LIN {X 0,Y 317.742,Z 934.096,A -85,B 0,C 180,E1 -15208.733,E2 -15208.733} C_VEL
LIN {X 0,Y 317.78,Z 934.392,A -85,B 0,C 180,E1 -15210,E2 -15210} C_VEL
LIN {X 0,Y 317.742,Z 934.092,A -85,B 0,C 180,E1 -15211.267,E2 -15211.267} C_VEL
LIN {X 0,Y 317.766,Z 933.304,A -85,B 0,C 180,E1 -15212.535,E2 -15212.535} C_VEL
LIN {X 0,Y 317.849,Z 932.043,A -85,B 0,C 180,E1 -15213.803,E2 -15213.803} C_VEL
LIN {X 0,Y 317.9,Z 930.281,A -85,B 0,C 180,E1 -15215.073,E2 -15215.073} C_VEL
LIN {X 0,Y 318.202,Z 926.465,A -85,B 0,C 180,E1 -15216.977,E2 -15216.977} C_VEL
LIN {X 0,Y 318.673,Z 921.267,A -85,B 0,C 180,E1 -15218.881,E2 -15218.881} C_VEL
LIN {X 0,Y 319.407,Z 914.42,A -85,B 0,C 180,E1 -15220.779,E2 -15220.779} C_VEL
LIN {X 0,Y 320.293,Z 906.941,A -85,B 0,C 180,E1 -15222.353,E2 -15222.353} C_VEL
LIN {X 0,Y 321.122,Z 899.567,A -85,B 0,C 180,E1 -15223.608,E2 -15223.608} C_VEL
LIN {X 0,Y 322.069,Z 891.674,A -85,B 0,C 180,E1 -15224.695,E2 -15224.695} C_VEL
LIN {X 0,Y 322.96,Z 883.333,A -85,B 0,C 180,E1 -15225.622,E2 -15225.622} C_VEL
LIN {X 0,Y 323.821,Z 872.672,A -85,B 0,C 180,E1 -15226.55,E2 -15226.55} C_VEL
LIN {X 0,Y 324.536,Z 861.891,A -85,B 0,C 180,E1 -15227.202,E2 -15227.202} C_VEL
LIN {X 0,Y 325.052,Z 852.616,A -85,B 0,C 180,E1 -15227.579,E2 -15227.579} C_VEL
LIN {X 0,Y 325.448,Z 824.387,A -85,B 0,C 180,E1 -15228.247,E2 -15228.247} C_VEL
LIN {X 0,Y 325.686,Z 806.284,A -85,B 0,C 180,E1 -15228.645,E2 -15228.645} C_VEL
LIN {X 0,Y 321.847,Z 779.896,A -85,B 0,C 180,E1 -15229.482,E2 -15229.482} C_VEL
LIN {X 0,Y 320.974,Z 774.315,A -85,B 0,C 180,E1 -15229.718,E2 -15229.718} C_VEL
LIN {X 0,Y 322.187,Z 763.095,A -85,B 0,C 180,E1 -15233.119,E2 -15233.119} C_VEL
LIN {X 0,Y 321.81,Z 758.821,A -85,B 0,C 180,E1 -15234.516,E2 -15234.516} C_VEL
LIN {X 0,Y 319.887,Z 748.827,A -85,B 0,C 180,E1 -15237.932,E2 -15237.932} C_VEL
LIN {X 0,Y 319.627,Z 747.504,A -85,B 0,C 180,E1 -15238.472,E2 -15238.472} C_VEL
LIN {X 0,Y 319.533,Z 747.475,A -85,B 0,C 180,E1 -15241.862,E2 -15241.862} C_VEL
LIN {X 0,Y 319.58,Z 747.478,A -85,B 0,C 180,E1 -15245.543,E2 -15245.543} C_VEL
LIN {X 0,Y 319.574,Z 747.49,A -85,B 0,C 180,E1 -15248.008,E2 -15248.008} C_VEL
LIN {X 0,Y 319.526,Z 747.474,A -85,B 0,C 180,E1 -15251.597,E2 -15251.597} C_VEL
LIN {X 0,Y 319.506,Z 747.499,A -85,B 0,C 180,E1 -15255.261,E2 -15255.261} C_VEL
LIN {X 0,Y 319.544,Z 747.457,A -85,B 0,C 180,E1 -15258.714,E2 -15258.714} C_VEL
LIN {X 0,Y 319.582,Z 747.448,A -85,B 0,C 180,E1 -15262.343,E2 -15262.343} C_VEL
LIN {X 0,Y 319.561,Z 747.485,A -85,B 0,C 180,E1 -15265.124,E2 -15265.124} C_VEL
LIN {X 0,Y 319.567,Z 747.483,A -85,B 0,C 180,E1 -15269.059,E2 -15269.059} C_VEL
LIN {X 0,Y 319.607,Z 747.482,A -85,B 0,C 180,E1 -15272.498,E2 -15272.498} C_VEL
LIN {X 0,Y 319.608,Z 747.484,A -85,B 0,C 180,E1 -15275.304,E2 -15275.304} C_VEL
LIN {X 0,Y 319.623,Z 747.463,A -85,B 0,C 180,E1 -15279.402,E2 -15279.402} C_VEL
LIN {X 0,Y 319.66,Z 747.478,A -85,B 0,C 180,E1 -15282.073,E2 -15282.073} C_VEL
LIN {X 0,Y 319.733,Z 747.455,A -85,B 0,C 180,E1 -15286.008,E2 -15286.008} C_VEL
LIN {X 0,Y 319.758,Z 747.454,A -85,B 0,C 180,E1 -15289.873,E2 -15289.873} C_VEL
LIN {X 0,Y 319.914,Z 747.45,A -85,B 0,C 180,E1 -15292.426,E2 -15292.426} C_VEL
LIN {X 0,Y 319.747,Z 747.458,A -85,B 0,C 180,E1 -15294.956,E2 -15294.956} C_VEL
LIN {X 0,Y 319.992,Z 747.407,A -85,B 0,C 180,E1 -15297.483,E2 -15297.483} C_VEL
LIN {X 0,Y 320.152,Z 747.405,A -85,B 0,C 180,E1 -15300,E2 -15300} C_VEL
LIN {X 0,Y 320.011,Z 747.437,A -85,B 0,C 180,E1 -15302.518,E2 -15302.518} C_VEL
LIN {X 0,Y 319.935,Z 747.42,A -85,B 0,C 180,E1 -15306.589,E2 -15306.589} C_VEL
LIN {X 0,Y 319.759,Z 747.456,A -85,B 0,C 180,E1 -15310.127,E2 -15310.127} C_VEL
LIN {X 0,Y 319.734,Z 747.466,A -85,B 0,C 180,E1 -15313.992,E2 -15313.992} C_VEL
LIN {X 0,Y 319.625,Z 747.462,A -85,B 0,C 180,E1 -15317.929,E2 -15317.929} C_VEL
LIN {X 0,Y 319.599,Z 747.483,A -85,B 0,C 180,E1 -15320.6,E2 -15320.6} C_VEL
LIN {X 0,Y 319.604,Z 747.472,A -85,B 0,C 180,E1 -15324.696,E2 -15324.696} C_VEL
LIN {X 0,Y 319.612,Z 747.479,A -85,B 0,C 180,E1 -15328.41,E2 -15328.41} C_VEL
LIN {X 0,Y 319.532,Z 747.486,A -85,B 0,C 180,E1 -15331.862,E2 -15331.862} C_VEL
LIN {X 0,Y 319.581,Z 747.487,A -85,B 0,C 180,E1 -15335.543,E2 -15335.543} C_VEL
LIN {X 0,Y 319.558,Z 747.487,A -85,B 0,C 180,E1 -15338.01,E2 -15338.01} C_VEL
LIN {X 0,Y 319.526,Z 747.448,A -85,B 0,C 180,E1 -15341.597,E2 -15341.597} C_VEL
LIN {X 0,Y 319.489,Z 747.484,A -85,B 0,C 180,E1 -15345.257,E2 -15345.257} C_VEL
LIN {X 0,Y 319.53,Z 747.494,A -85,B 0,C 180,E1 -15348.712,E2 -15348.712} C_VEL
LIN {X 0,Y 319.555,Z 747.468,A -85,B 0,C 180,E1 -15352.35,E2 -15352.35} C_VEL
LIN {X 0,Y 319.561,Z 747.494,A -85,B 0,C 180,E1 -15355.124,E2 -15355.124} C_VEL
LIN {X 0,Y 319.525,Z 747.479,A -85,B 0,C 180,E1 -15358.137,E2 -15358.137} C_VEL
LIN {X 0,Y 319.573,Z 747.488,A -85,B 0,C 180,E1 -15361.603,E2 -15361.603} C_VEL
LIN {X 0,Y 319.58,Z 747.491,A -85,B 0,C 180,E1 -15365.302,E2 -15365.302} C_VEL
LIN {X 0,Y 319.648,Z 747.739,A -85,B 0,C 180,E1 -15366.787,E2 -15366.787} C_VEL
LIN {X 0,Y 320.884,Z 754.66,A -85,B 0,C 180,E1 -15369.486,E2 -15369.486} C_VEL
LIN {X 0,Y 321.16,Z 757.232,A -85,B 0,C 180,E1 -15370.352,E2 -15370.352} C_VEL
LIN {X 0,Y 322.337,Z 762.306,A -85,B 0,C 180,E1 -15370.6,E2 -15370.6} C_VEL
LIN {X 0,Y 326.157,Z 782.212,A -85,B 0,C 180,E1 -15371.294,E2 -15371.294} C_VEL
LIN {X 0,Y 325.308,Z 832.933,A -85,B 0,C 180,E1 -15372.435,E2 -15372.435} C_VEL
LIN {X 0,Y 325.067,Z 841.877,A -85,B 0,C 180,E1 -15372.787,E2 -15372.787} C_VEL
LIN {X 0,Y 324.487,Z 851.397,A -85,B 0,C 180,E1 -15373.323,E2 -15373.323} C_VEL
LIN {X 0,Y 323.868,Z 859.523,A -85,B 0,C 180,E1 -15373.938,E2 -15373.938} C_VEL
LIN {X 0,Y 323.181,Z 867.591,A -85,B 0,C 180,E1 -15374.712,E2 -15374.712} C_VEL
LIN {X 0,Y 322.335,Z 876.66,A -85,B 0,C 180,E1 -15375.801,E2 -15375.801} C_VEL
LIN {X 0,Y 321.439,Z 884.87,A -85,B 0,C 180,E1 -15377.05,E2 -15377.05} C_VEL
LIN {X 0,Y 320.62,Z 891.505,A -85,B 0,C 180,E1 -15378.302,E2 -15378.302} C_VEL
LIN {X 0,Y 319.731,Z 898.19,A -85,B 0,C 180,E1 -15379.872,E2 -15379.872} C_VEL
LIN {X 0,Y 319.197,Z 902.589,A -85,B 0,C 180,E1 -15381.134,E2 -15381.134} C_VEL
LIN {X 0,Y 318.638,Z 907.674,A -85,B 0,C 180,E1 -15382.997,E2 -15382.997} C_VEL
LIN {X 0,Y 318.381,Z 910.411,A -85,B 0,C 180,E1 -15384.299,E2 -15384.299} C_VEL
LIN {X 0,Y 318.03,Z 913.317,A -85,B 0,C 180,E1 -15386.199,E2 -15386.199} C_VEL
LIN {X 0,Y 317.874,Z 914.586,A -85,B 0,C 180,E1 -15387.466,E2 -15387.466} C_VEL
LIN {X 0,Y 317.791,Z 915.386,A -85,B 0,C 180,E1 -15388.733,E2 -15388.733} C_VEL
LIN {X 0,Y 317.787,Z 915.69,A -85,B 0,C 180,E1 -15390,E2 -15390} C_VEL
LIN {X 0,Y 317.789,Z 915.413,A -85,B 0,C 180,E1 -15391.267,E2 -15391.267} C_VEL
LIN {X 0,Y 317.865,Z 914.667,A -85,B 0,C 180,E1 -15392.534,E2 -15392.534} C_VEL
LIN {X 0,Y 318.029,Z 913.452,A -85,B 0,C 180,E1 -15393.801,E2 -15393.801} C_VEL
LIN {X 0,Y 318.366,Z 910.603,A -85,B 0,C 180,E1 -15395.701,E2 -15395.701} C_VEL
LIN {X 0,Y 318.633,Z 907.943,A -85,B 0,C 180,E1 -15396.996,E2 -15396.996} C_VEL
LIN {X 0,Y 319.144,Z 902.909,A -85,B 0,C 180,E1 -15398.868,E2 -15398.868} C_VEL
LIN {X 0,Y 319.815,Z 897.417,A -85,B 0,C 180,E1 -15400.445,E2 -15400.445} C_VEL
LIN {X 0,Y 320.722,Z 890.511,A -85,B 0,C 180,E1 -15402.015,E2 -15402.015} C_VEL
LIN {X 0,Y 321.68,Z 882.579,A -85,B 0,C 180,E1 -15403.423,E2 -15403.423} C_VEL
LIN {X 0,Y 322.502,Z 875.014,A -85,B 0,C 180,E1 -15404.514,E2 -15404.514} C_VEL
LIN {X 0,Y 323.321,Z 867.081,A -85,B 0,C 180,E1 -15405.443,E2 -15405.443} C_VEL
LIN {X 0,Y 324.015,Z 858.885,A -85,B 0,C 180,E1 -15406.216,E2 -15406.216} C_VEL
LIN {X 0,Y 324.615,Z 850.571,A -85,B 0,C 180,E1 -15406.832,E2 -15406.832} C_VEL
LIN {X 0,Y 325.054,Z 841.576,A -85,B 0,C 180,E1 -15407.335,E2 -15407.335} C_VEL
LIN {X 0,Y 325.37,Z 831.849,A -85,B 0,C 180,E1 -15407.702,E2 -15407.702} C_VEL
LIN {X 0,Y 326.103,Z 781.764,A -85,B 0,C 180,E1 -15408.827,E2 -15408.827} C_VEL
LIN {X 0,Y 321.94,Z 760.624,A -85,B 0,C 180,E1 -15409.573,E2 -15409.573} C_VEL
LIN {X 0,Y 321.097,Z 756.993,A -85,B 0,C 180,E1 -15409.752,E2 -15409.752} C_VEL
LIN {X 0,Y 320.184,Z 750.297,A -85,B 0,C 180,E1 -15412.302,E2 -15412.302} C_VEL
LIN {X 0,Y 319.64,Z 747.554,A -85,B 0,C 180,E1 -15413.486,E2 -15413.486} C_VEL
LIN {X 0,Y 319.546,Z 747.492,A -85,B 0,C 180,E1 -15417.508,E2 -15417.508} C_VEL
LIN {X 0,Y 319.55,Z 747.481,A -85,B 0,C 180,E1 -15420.936,E2 -15420.936} C_VEL
LIN {X 0,Y 319.577,Z 747.486,A -85,B 0,C 180,E1 -15423.353,E2 -15423.353} C_VEL
LIN {X 0,Y 319.559,Z 747.484,A -85,B 0,C 180,E1 -15426.428,E2 -15426.428} C_VEL
LIN {X 0,Y 319.56,Z 747.472,A -85,B 0,C 180,E1 -15429.669,E2 -15429.669} C_VEL
LIN {X 0,Y 319.523,Z 747.493,A -85,B 0,C 180,E1 -15433.461,E2 -15433.461} C_VEL
LIN {X 0,Y 319.485,Z 747.489,A -85,B 0,C 180,E1 -15434.127,E2 -15434.127} C_VEL
LIN {X 0,Y 318.807,Z 747.567,A -85,B 0,C 180,E1 -15435.18,E2 -15435.18} C_VEL
LIN {X 0,Y 315.957,Z 747.898,A -85,B 0,C 180,E1 -15436.895,E2 -15436.895} C_VEL
LIN {X 0,Y 313.566,Z 748.191,A -85,B 0,C 180,E1 -15438.285,E2 -15438.285} C_VEL
LIN {X 0,Y 312.566,Z 748.328,A -85,B 0,C 180,E1 -15439.361,E2 -15439.361} C_VEL
LIN {X 0,Y 312.498,Z 748.344,A -85,B 0,C 180,E1 -15439.725,E2 -15439.725} C_VEL
LIN {X 0,Y 312.527,Z 748.367,A -85,B 0,C 180,E1 -15442.615,E2 -15442.615} C_VEL
LIN {X 0,Y 312.52,Z 748.354,A -85,B 0,C 180,E1 -15446.311,E2 -15446.311} C_VEL
LIN {X 0,Y 312.539,Z 748.365,A -85,B 0,C 180,E1 -15450.349,E2 -15450.349} C_VEL
LIN {X 0,Y 312.598,Z 748.336,A -85,B 0,C 180,E1 -15454.067,E2 -15454.067} C_VEL
LIN {X 0,Y 312.566,Z 748.362,A -85,B 0,C 180,E1 -15457.527,E2 -15457.527} C_VEL
LIN {X 0,Y 312.59,Z 748.34,A -85,B 0,C 180,E1 -15461.653,E2 -15461.653} C_VEL
LIN {X 0,Y 312.687,Z 748.345,A -85,B 0,C 180,E1 -15465.686,E2 -15465.686} C_VEL
LIN {X 0,Y 312.704,Z 748.337,A -85,B 0,C 180,E1 -15469.642,E2 -15469.642} C_VEL
LIN {X 0,Y 312.873,Z 748.294,A -85,B 0,C 180,E1 -15472.254,E2 -15472.254} C_VEL
LIN {X 0,Y 312.72,Z 748.331,A -85,B 0,C 180,E1 -15474.842,E2 -15474.842} C_VEL
LIN {X 0,Y 312.954,Z 748.316,A -85,B 0,C 180,E1 -15477.426,E2 -15477.426} C_VEL
LIN {X 0,Y 313.103,Z 748.283,A -85,B 0,C 180,E1 -15480,E2 -15480} C_VEL
LIN {X 0,Y 312.938,Z 748.286,A -85,B 0,C 180,E1 -15482.574,E2 -15482.574} C_VEL
LIN {X 0,Y 312.902,Z 748.318,A -85,B 0,C 180,E1 -15486.448,E2 -15486.448} C_VEL
LIN {X 0,Y 312.787,Z 748.332,A -85,B 0,C 180,E1 -15489.049,E2 -15489.049} C_VEL
LIN {X 0,Y 312.635,Z 748.33,A -85,B 0,C 180,E1 -15492.991,E2 -15492.991} C_VEL
LIN {X 0,Y 312.64,Z 748.35,A -85,B 0,C 180,E1 -15495.65,E2 -15495.65} C_VEL
LIN {X 0,Y 312.608,Z 748.344,A -85,B 0,C 180,E1 -15499.708,E2 -15499.708} C_VEL
LIN {X 0,Y 312.548,Z 748.354,A -85,B 0,C 180,E1 -15502.79,E2 -15502.79} C_VEL
LIN {X 0,Y 312.603,Z 748.361,A -85,B 0,C 180,E1 -15505.935,E2 -15505.935} C_VEL
LIN {X 0,Y 312.538,Z 748.347,A -85,B 0,C 180,E1 -15509.65,E2 -15509.65} C_VEL
LIN {X 0,Y 312.52,Z 748.369,A -85,B 0,C 180,E1 -15513.689,E2 -15513.689} C_VEL
LIN {X 0,Y 312.541,Z 748.328,A -85,B 0,C 180,E1 -15517.383,E2 -15517.383} C_VEL
LIN {X 0,Y 312.5,Z 748.323,A -85,B 0,C 180,E1 -15520.707,E2 -15520.707} C_VEL
LIN {X 0,Y 312.471,Z 748.373,A -85,B 0,C 180,E1 -15524.206,E2 -15524.206} C_VEL
LIN {X 0,Y 312.485,Z 748.352,A -85,B 0,C 180,E1 -15527.918,E2 -15527.918} C_VEL
LIN {X 0,Y 312.536,Z 748.367,A -85,B 0,C 180,E1 -15531.91,E2 -15531.91} C_VEL
LIN {X 0,Y 312.507,Z 748.37,A -85,B 0,C 180,E1 -15535.79,E2 -15535.79} C_VEL
LIN {X 0,Y 312.524,Z 748.338,A -85,B 0,C 180,E1 -15538.854,E2 -15538.854} C_VEL
LIN {X 0,Y 312.59,Z 748.504,A -85,B 0,C 180,E1 -15541.264,E2 -15541.264} C_VEL
LIN {X 0,Y 314.23,Z 756.797,A -85,B 0,C 180,E1 -15544.233,E2 -15544.233} C_VEL
LIN {X 0,Y 315.221,Z 762.929,A -85,B 0,C 180,E1 -15546.339,E2 -15546.339} C_VEL
LIN {X 0,Y 314.425,Z 770.35,A -85,B 0,C 180,E1 -15548.702,E2 -15548.702} C_VEL
LIN {X 0,Y 314.084,Z 774.254,A -85,B 0,C 180,E1 -15549.828,E2 -15549.828} C_VEL
LIN {X 0,Y 317.45,Z 795.547,A -85,B 0,C 180,E1 -15550.589,E2 -15550.589} C_VEL
LIN {X 0,Y 319.097,Z 808.819,A -85,B 0,C 180,E1 -15551.001,E2 -15551.001} C_VEL
LIN {X 0,Y 318.357,Z 851.659,A -85,B 0,C 180,E1 -15551.997,E2 -15551.997} C_VEL
LIN {X 0,Y 317.733,Z 862.861,A -85,B 0,C 180,E1 -15552.46,E2 -15552.46} C_VEL
LIN {X 0,Y 316.855,Z 874.578,A -85,B 0,C 180,E1 -15553.241,E2 -15553.241} C_VEL
LIN {X 0,Y 316.106,Z 883.279,A -85,B 0,C 180,E1 -15554.03,E2 -15554.03} C_VEL
LIN {X 0,Y 315.185,Z 891.589,A -85,B 0,C 180,E1 -15554.977,E2 -15554.977} C_VEL
LIN {X 0,Y 314.229,Z 899.457,A -85,B 0,C 180,E1 -15556.088,E2 -15556.088} C_VEL
LIN {X 0,Y 313.339,Z 906.817,A -85,B 0,C 180,E1 -15557.368,E2 -15557.368} C_VEL
LIN {X 0,Y 312.432,Z 914.287,A -85,B 0,C 180,E1 -15558.977,E2 -15558.977} C_VEL
LIN {X 0,Y 311.641,Z 921.109,A -85,B 0,C 180,E1 -15560.917,E2 -15560.917} C_VEL
LIN {X 0,Y 311.128,Z 926.294,A -85,B 0,C 180,E1 -15562.863,E2 -15562.863} C_VEL
LIN {X 0,Y 310.819,Z 930.102,A -85,B 0,C 180,E1 -15564.811,E2 -15564.811} C_VEL
LIN {X 0,Y 310.762,Z 931.855,A -85,B 0,C 180,E1 -15566.11,E2 -15566.11} C_VEL
LIN {X 0,Y 310.69,Z 933.109,A -85,B 0,C 180,E1 -15567.407,E2 -15567.407} C_VEL
LIN {X 0,Y 310.657,Z 933.888,A -85,B 0,C 180,E1 -15568.704,E2 -15568.704} C_VEL
LIN {X 0,Y 310.69,Z 934.184,A -85,B 0,C 180,E1 -15570,E2 -15570} C_VEL
LIN {X 0,Y 310.657,Z 933.884,A -85,B 0,C 180,E1 -15571.296,E2 -15571.296} C_VEL
LIN {X 0,Y 310.69,Z 933.096,A -85,B 0,C 180,E1 -15572.593,E2 -15572.593} C_VEL
LIN {X 0,Y 310.762,Z 931.833,A -85,B 0,C 180,E1 -15573.89,E2 -15573.89} C_VEL
LIN {X 0,Y 310.894,Z 928.751,A -85,B 0,C 180,E1 -15575.929,E2 -15575.929} C_VEL
LIN {X 0,Y 311.254,Z 924.727,A -85,B 0,C 180,E1 -15577.786,E2 -15577.786} C_VEL
LIN {X 0,Y 311.846,Z 919.003,A -85,B 0,C 180,E1 -15579.731,E2 -15579.731} C_VEL
LIN {X 0,Y 312.59,Z 912.791,A -85,B 0,C 180,E1 -15581.346,E2 -15581.346} C_VEL
LIN {X 0,Y 313.338,Z 906.729,A -85,B 0,C 180,E1 -15582.632,E2 -15582.632} C_VEL
LIN {X 0,Y 314.213,Z 899.354,A -85,B 0,C 180,E1 -15583.913,E2 -15583.913} C_VEL
LIN {X 0,Y 315.207,Z 891.461,A -85,B 0,C 180,E1 -15585.022,E2 -15585.022} C_VEL
LIN {X 0,Y 316.13,Z 883.119,A -85,B 0,C 180,E1 -15585.969,E2 -15585.969} C_VEL
LIN {X 0,Y 317.009,Z 872.456,A -85,B 0,C 180,E1 -15586.917,E2 -15586.917} C_VEL
LIN {X 0,Y 317.837,Z 860.841,A -85,B 0,C 180,E1 -15587.617,E2 -15587.617} C_VEL
LIN {X 0,Y 318.335,Z 851.094,A -85,B 0,C 180,E1 -15588.004,E2 -15588.004} C_VEL
LIN {X 0,Y 318.986,Z 807.307,A -85,B 0,C 180,E1 -15589.022,E2 -15589.022} C_VEL
LIN {X 0,Y 315.441,Z 782.581,A -85,B 0,C 180,E1 -15589.826,E2 -15589.826} C_VEL
LIN {X 0,Y 314.063,Z 774.36,A -85,B 0,C 180,E1 -15590.141,E2 -15590.141} C_VEL
LIN {X 0,Y 314.096,Z 773.321,A -85,B 0,C 180,E1 -15590.356,E2 -15590.356} C_VEL
LIN {X 0,Y 315.211,Z 763.954,A -85,B 0,C 180,E1 -15593.313,E2 -15593.313} C_VEL
LIN {X 0,Y 314.577,Z 758.61,A -85,B 0,C 180,E1 -15595.118,E2 -15595.118} C_VEL
LIN {X 0,Y 312.74,Z 749.169,A -85,B 0,C 180,E1 -15598.439,E2 -15598.439} C_VEL
LIN {X 0,Y 312.577,Z 748.373,A -85,B 0,C 180,E1 -15598.864,E2 -15598.864} C_VEL
LIN {X 0,Y 312.505,Z 748.364,A -85,B 0,C 180,E1 -15602.666,E2 -15602.666} C_VEL
LIN {X 0,Y 312.536,Z 748.355,A -85,B 0,C 180,E1 -15605.95,E2 -15605.95} C_VEL
LIN {X 0,Y 312.508,Z 748.368,A -85,B 0,C 180,E1 -15609.027,E2 -15609.027} C_VEL
LIN {X 0,Y 312.492,Z 748.356,A -85,B 0,C 180,E1 -15612.431,E2 -15612.431} C_VEL
LIN {X 0,Y 312.483,Z 748.369,A -85,B 0,C 180,E1 -15616.03,E2 -15616.03} C_VEL
LIN {X 0,Y 312.5,Z 748.321,A -85,B 0,C 180,E1 -15619.293,E2 -15619.293} C_VEL
LIN {X 0,Y 312.541,Z 748.33,A -85,B 0,C 180,E1 -15622.617,E2 -15622.617} C_VEL
LIN {X 0,Y 312.52,Z 748.369,A -85,B 0,C 180,E1 -15626.311,E2 -15626.311} C_VEL
LIN {X 0,Y 312.538,Z 748.347,A -85,B 0,C 180,E1 -15630.35,E2 -15630.35} C_VEL
LIN {X 0,Y 312.603,Z 748.361,A -85,B 0,C 180,E1 -15634.065,E2 -15634.065} C_VEL
LIN {X 0,Y 312.589,Z 748.344,A -85,B 0,C 180,E1 -15637.529,E2 -15637.529} C_VEL
LIN {X 0,Y 312.64,Z 748.348,A -85,B 0,C 180,E1 -15641.657,E2 -15641.657} C_VEL
LIN {X 0,Y 312.695,Z 748.336,A -85,B 0,C 180,E1 -15645.686,E2 -15645.686} C_VEL
LIN {X 0,Y 312.702,Z 748.331,A -85,B 0,C 180,E1 -15649.642,E2 -15649.642} C_VEL
LIN {X 0,Y 312.855,Z 748.328,A -85,B 0,C 180,E1 -15652.254,E2 -15652.254} C_VEL
LIN {X 0,Y 312.717,Z 748.334,A -85,B 0,C 180,E1 -15654.843,E2 -15654.843} C_VEL
LIN {X 0,Y 312.992,Z 748.285,A -85,B 0,C 180,E1 -15658.714,E2 -15658.714} C_VEL
LIN {X 0,Y 312.994,Z 748.305,A -85,B 0,C 180,E1 -15661.287,E2 -15661.287} C_VEL
LIN {X 0,Y 312.698,Z 748.343,A -85,B 0,C 180,E1 -15663.866,E2 -15663.866} C_VEL
LIN {X 0,Y 312.901,Z 748.296,A -85,B 0,C 180,E1 -15666.57,E2 -15666.57} C_VEL
LIN {X 0,Y 312.789,Z 748.315,A -85,B 0,C 180,E1 -15669.049,E2 -15669.049} C_VEL
LIN {X 0,Y 312.636,Z 748.354,A -85,B 0,C 180,E1 -15672.991,E2 -15672.991} C_VEL
LIN {X 0,Y 312.626,Z 748.34,A -85,B 0,C 180,E1 -15675.65,E2 -15675.65} C_VEL
LIN {X 0,Y 312.566,Z 748.357,A -85,B 0,C 180,E1 -15679.711,E2 -15679.711} C_VEL
LIN {X 0,Y 312.527,Z 748.367,A -85,B 0,C 180,E1 -15682.781,E2 -15682.781} C_VEL
LIN {X 0,Y 312.598,Z 748.336,A -85,B 0,C 180,E1 -15685.933,E2 -15685.933} C_VEL
LIN {X 0,Y 312.539,Z 748.365,A -85,B 0,C 180,E1 -15689.651,E2 -15689.651} C_VEL
LIN {X 0,Y 312.52,Z 748.353,A -85,B 0,C 180,E1 -15693.689,E2 -15693.689} C_VEL
LIN {X 0,Y 312.527,Z 748.368,A -85,B 0,C 180,E1 -15697.385,E2 -15697.385} C_VEL
LIN {X 0,Y 312.49,Z 748.338,A -85,B 0,C 180,E1 -15700.709,E2 -15700.709} C_VEL
LIN {X 0,Y 312.452,Z 748.341,A -85,B 0,C 180,E1 -15704.21,E2 -15704.21} C_VEL
LIN {X 0,Y 312.485,Z 748.373,A -85,B 0,C 180,E1 -15707.919,E2 -15707.919} C_VEL
LIN {X 0,Y 312.499,Z 748.346,A -85,B 0,C 180,E1 -15710.971,E2 -15710.971} C_VEL
LIN {X 0,Y 312.533,Z 748.367,A -85,B 0,C 180,E1 -15714.22,E2 -15714.22} C_VEL
LIN {X 0,Y 312.502,Z 748.358,A -85,B 0,C 180,E1 -15717.334,E2 -15717.334} C_VEL
LIN {X 0,Y 312.508,Z 748.37,A -85,B 0,C 180,E1 -15721.291,E2 -15721.291} C_VEL
LIN {X 0,Y 312.551,Z 748.364,A -85,B 0,C 180,E1 -15724.708,E2 -15724.708} C_VEL
LIN {X 0,Y 312.556,Z 748.465,A -85,B 0,C 180,E1 -15726.405,E2 -15726.405} C_VEL
LIN {X 0,Y 313.772,Z 754.871,A -85,B 0,C 180,E1 -15729,E2 -15729} C_VEL
LIN {X 0,Y 314.097,Z 757.359,A -85,B 0,C 180,E1 -15729.877,E2 -15729.877} C_VEL
LIN {X 0,Y 315.025,Z 760.896,A -85,B 0,C 180,E1 -15730.091,E2 -15730.091} C_VEL
LIN {X 0,Y 318.72,Z 778.989,A -85,B 0,C 180,E1 -15730.759,E2 -15730.759} C_VEL
LIN {X 0,Y 319.417,Z 784.32,A -85,B 0,C 180,E1 -15730.928,E2 -15730.928} C_VEL
LIN {X 0,Y 318.558,Z 833.159,A -85,B 0,C 180,E1 -15732.051,E2 -15732.051} C_VEL
LIN {X 0,Y 318.306,Z 842.097,A -85,B 0,C 180,E1 -15732.41,E2 -15732.41} C_VEL
LIN {X 0,Y 317.722,Z 851.613,A -85,B 0,C 180,E1 -15732.957,E2 -15732.957} C_VEL
LIN {X 0,Y 317.061,Z 859.738,A -85,B 0,C 180,E1 -15733.583,E2 -15733.583} C_VEL
LIN {X 0,Y 316.361,Z 867.805,A -85,B 0,C 180,E1 -15734.374,E2 -15734.374} C_VEL
LIN {X 0,Y 315.474,Z 876.873,A -85,B 0,C 180,E1 -15735.486,E2 -15735.486} C_VEL
LIN {X 0,Y 314.538,Z 885.082,A -85,B 0,C 180,E1 -15736.76,E2 -15736.76} C_VEL
LIN {X 0,Y 313.682,Z 891.716,A -85,B 0,C 180,E1 -15738.039,E2 -15738.039} C_VEL
LIN {X 0,Y 312.74,Z 898.401,A -85,B 0,C 180,E1 -15739.643,E2 -15739.643} C_VEL
LIN {X 0,Y 312.197,Z 902.799,A -85,B 0,C 180,E1 -15740.934,E2 -15740.934} C_VEL
LIN {X 0,Y 311.829,Z 906.458,A -85,B 0,C 180,E1 -15742.228,E2 -15742.228} C_VEL
LIN {X 0,Y 311.419,Z 909.451,A -85,B 0,C 180,E1 -15743.521,E2 -15743.521} C_VEL
LIN {X 0,Y 311.207,Z 911.765,A -85,B 0,C 180,E1 -15744.817,E2 -15744.817} C_VEL
LIN {X 0,Y 310.969,Z 913.526,A -85,B 0,C 180,E1 -15746.112,E2 -15746.112} C_VEL
LIN {X 0,Y 310.797,Z 914.795,A -85,B 0,C 180,E1 -15747.408,E2 -15747.408} C_VEL
LIN {X 0,Y 310.705,Z 915.595,A -85,B 0,C 180,E1 -15748.704,E2 -15748.704} C_VEL
LIN {X 0,Y 310.697,Z 915.899,A -85,B 0,C 180,E1 -15750,E2 -15750} C_VEL
LIN {X 0,Y 310.703,Z 915.621,A -85,B 0,C 180,E1 -15751.296,E2 -15751.296} C_VEL
LIN {X 0,Y 310.789,Z 914.875,A -85,B 0,C 180,E1 -15752.592,E2 -15752.592} C_VEL
LIN {X 0,Y 310.967,Z 913.659,A -85,B 0,C 180,E1 -15753.888,E2 -15753.888} C_VEL
LIN {X 0,Y 311.31,Z 910.81,A -85,B 0,C 180,E1 -15755.831,E2 -15755.831} C_VEL
LIN {X 0,Y 311.542,Z 908.559,A -85,B 0,C 180,E1 -15756.98,E2 -15756.98} C_VEL
LIN {X 0,Y 311.933,Z 905.017,A -85,B 0,C 180,E1 -15758.421,E2 -15758.421} C_VEL
LIN {X 0,Y 312.532,Z 899.958,A -85,B 0,C 180,E1 -15760.037,E2 -15760.037} C_VEL
LIN {X 0,Y 313.225,Z 895.01,A -85,B 0,C 180,E1 -15761.322,E2 -15761.322} C_VEL
LIN {X 0,Y 314.023,Z 889.037,A -85,B 0,C 180,E1 -15762.604,E2 -15762.604} C_VEL
LIN {X 0,Y 314.878,Z 881.767,A -85,B 0,C 180,E1 -15763.883,E2 -15763.883} C_VEL
LIN {X 0,Y 315.615,Z 875.22,A -85,B 0,C 180,E1 -15764.837,E2 -15764.837} C_VEL
LIN {X 0,Y 316.501,Z 867.285,A -85,B 0,C 180,E1 -15765.784,E2 -15765.784} C_VEL
LIN {X 0,Y 317.228,Z 859.086,A -85,B 0,C 180,E1 -15766.573,E2 -15766.573} C_VEL
LIN {X 0,Y 317.854,Z 850.77,A -85,B 0,C 180,E1 -15767.201,E2 -15767.201} C_VEL
LIN {X 0,Y 318.304,Z 841.773,A -85,B 0,C 180,E1 -15767.715,E2 -15767.715} C_VEL
LIN {X 0,Y 318.601,Z 832.212,A -85,B 0,C 180,E1 -15768.086,E2 -15768.086} C_VEL
LIN {X 0,Y 319.415,Z 782.769,A -85,B 0,C 180,E1 -15769.217,E2 -15769.217} C_VEL
LIN {X 0,Y 315.595,Z 763.033,A -85,B 0,C 180,E1 -15769.93,E2 -15769.93} C_VEL
LIN {X 0,Y 314.117,Z 757.566,A -85,B 0,C 180,E1 -15770.203,E2 -15770.203} C_VEL
LIN {X 0,Y 314.014,Z 756.765,A -85,B 0,C 180,E1 -15770.39,E2 -15770.39} C_VEL
LIN {X 0,Y 312.769,Z 749.315,A -85,B 0,C 180,E1 -15773.322,E2 -15773.322} C_VEL
LIN {X 0,Y 312.591,Z 748.449,A -85,B 0,C 180,E1 -15773.738,E2 -15773.738} C_VEL
LIN {X 0,Y 312.498,Z 748.373,A -85,B 0,C 180,E1 -15776.731,E2 -15776.731} C_VEL
LIN {X 0,Y 312.497,Z 748.372,A -85,B 0,C 180,E1 -15779.655,E2 -15779.655} C_VEL
LIN {X 0,Y 312.521,Z 748.366,A -85,B 0,C 180,E1 -15783.689,E2 -15783.689} C_VEL
LIN {X 0,Y 312.521,Z 748.349,A -85,B 0,C 180,E1 -15787.386,E2 -15787.386} C_VEL
LIN {X 0,Y 312.491,Z 748.362,A -85,B 0,C 180,E1 -15790.709,E2 -15790.709} C_VEL
LIN {X 0,Y 312.453,Z 748.369,A -85,B 0,C 180,E1 -15794.21,E2 -15794.21} C_VEL
LIN {X 0,Y 312.485,Z 748.32,A -85,B 0,C 180,E1 -15797.919,E2 -15797.919} C_VEL
LIN {X 0,Y 312.498,Z 748.344,A -85,B 0,C 180,E1 -15799.725,E2 -15799.725} C_VEL
LIN {X 0,Y 311.862,Z 748.444,A -85,B 0,C 180,E1 -15800.801,E2 -15800.801} C_VEL
LIN {X 0,Y 309.008,Z 748.81,A -85,B 0,C 180,E1 -15802.553,E2 -15802.553} C_VEL
LIN {X 0,Y 306.572,Z 749.108,A -85,B 0,C 180,E1 -15803.974,E2 -15803.974} C_VEL
LIN {X 0,Y 305.533,Z 749.231,A -85,B 0,C 180,E1 -15805.075,E2 -15805.075} C_VEL
LIN {X 0,Y 305.452,Z 749.238,A -85,B 0,C 180,E1 -15805.448,E2 -15805.448} C_VEL
LIN {X 0,Y 305.46,Z 749.247,A -85,B 0,C 180,E1 -15809.59,E2 -15809.59} C_VEL
LIN {X 0,Y 305.516,Z 749.23,A -85,B 0,C 180,E1 -15812.608,E2 -15812.608} C_VEL
LIN {X 0,Y 305.506,Z 749.229,A -85,B 0,C 180,E1 -15815.538,E2 -15815.538} C_VEL
LIN {X 0,Y 305.507,Z 749.237,A -85,B 0,C 180,E1 -15819.814,E2 -15819.814} C_VEL
LIN {X 0,Y 305.548,Z 749.213,A -85,B 0,C 180,E1 -15822.601,E2 -15822.601} C_VEL
LIN {X 0,Y 305.628,Z 749.219,A -85,B 0,C 180,E1 -15825.348,E2 -15825.348} C_VEL
LIN {X 0,Y 305.64,Z 749.219,A -85,B 0,C 180,E1 -15829.4,E2 -15829.4} C_VEL
LIN {X 0,Y 305.814,Z 749.173,A -85,B 0,C 180,E1 -15832.074,E2 -15832.074} C_VEL
LIN {X 0,Y 305.691,Z 749.206,A -85,B 0,C 180,E1 -15834.723,E2 -15834.723} C_VEL
LIN {X 0,Y 305.961,Z 749.181,A -85,B 0,C 180,E1 -15838.684,E2 -15838.684} C_VEL
LIN {X 0,Y 305.957,Z 749.161,A -85,B 0,C 180,E1 -15841.316,E2 -15841.316} C_VEL
LIN {X 0,Y 305.688,Z 749.211,A -85,B 0,C 180,E1 -15845.276,E2 -15845.276} C_VEL
LIN {X 0,Y 305.798,Z 749.205,A -85,B 0,C 180,E1 -15847.926,E2 -15847.926} C_VEL
LIN {X 0,Y 305.604,Z 749.203,A -85,B 0,C 180,E1 -15851.945,E2 -15851.945} C_VEL
LIN {X 0,Y 305.639,Z 749.218,A -85,B 0,C 180,E1 -15855.035,E2 -15855.035} C_VEL
LIN {X 0,Y 305.582,Z 749.223,A -85,B 0,C 180,E1 -15859.447,E2 -15859.447} C_VEL
LIN {X 0,Y 305.493,Z 749.233,A -85,B 0,C 180,E1 -15863.042,E2 -15863.042} C_VEL
LIN {X 0,Y 305.532,Z 749.238,A -85,B 0,C 180,E1 -15866.221,E2 -15866.221} C_VEL
LIN {X 0,Y 305.488,Z 749.225,A -85,B 0,C 180,E1 -15869.047,E2 -15869.047} C_VEL
LIN {X 0,Y 305.443,Z 749.247,A -85,B 0,C 180,E1 -15871.952,E2 -15871.952} C_VEL
LIN {X 0,Y 305.464,Z 749.239,A -85,B 0,C 180,E1 -15875.113,E2 -15875.113} C_VEL
LIN {X 0,Y 305.482,Z 749.188,A -85,B 0,C 180,E1 -15878.536,E2 -15878.536} C_VEL
LIN {X 0,Y 305.488,Z 749.228,A -85,B 0,C 180,E1 -15882.592,E2 -15882.592} C_VEL
LIN {X 0,Y 305.438,Z 749.243,A -85,B 0,C 180,E1 -15886.347,E2 -15886.347} C_VEL
LIN {X 0,Y 305.458,Z 749.234,A -85,B 0,C 180,E1 -15889.892,E2 -15889.892} C_VEL
LIN {X 0,Y 305.5,Z 749.232,A -85,B 0,C 180,E1 -15893.627,E2 -15893.627} C_VEL
LIN {X 0,Y 305.465,Z 749.249,A -85,B 0,C 180,E1 -15896.483,E2 -15896.483} C_VEL
LIN {X 0,Y 305.57,Z 749.392,A -85,B 0,C 180,E1 -15900.925,E2 -15900.925} C_VEL
LIN {X 0,Y 307.332,Z 758.46,A -85,B 0,C 180,E1 -15904.247,E2 -15904.247} C_VEL
LIN {X 0,Y 308.259,Z 764.978,A -85,B 0,C 180,E1 -15906.525,E2 -15906.525} C_VEL
LIN {X 0,Y 307.184,Z 773.882,A -85,B 0,C 180,E1 -15909.334,E2 -15909.334} C_VEL
LIN {X 0,Y 308.229,Z 779.909,A -85,B 0,C 180,E1 -15909.61,E2 -15909.61} C_VEL
LIN {X 0,Y 311.835,Z 804.283,A -85,B 0,C 180,E1 -15910.438,E2 -15910.438} C_VEL
LIN {X 0,Y 312.381,Z 811.143,A -85,B 0,C 180,E1 -15910.637,E2 -15910.637} C_VEL
LIN {X 0,Y 311.609,Z 851.465,A -85,B 0,C 180,E1 -15911.594,E2 -15911.594} C_VEL
LIN {X 0,Y 310.986,Z 862.662,A -85,B 0,C 180,E1 -15912.067,E2 -15912.067} C_VEL
LIN {X 0,Y 310.066,Z 874.374,A -85,B 0,C 180,E1 -15912.863,E2 -15912.863} C_VEL
LIN {X 0,Y 309.293,Z 883.075,A -85,B 0,C 180,E1 -15913.668,E2 -15913.668} C_VEL
LIN {X 0,Y 308.331,Z 891.384,A -85,B 0,C 180,E1 -15914.634,E2 -15914.634} C_VEL
LIN {X 0,Y 307.341,Z 899.251,A -85,B 0,C 180,E1 -15915.77,E2 -15915.77} C_VEL
LIN {X 0,Y 306.398,Z 906.61,A -85,B 0,C 180,E1 -15917.077,E2 -15917.077} C_VEL
LIN {X 0,Y 305.441,Z 914.079,A -85,B 0,C 180,E1 -15918.721,E2 -15918.721} C_VEL
LIN {X 0,Y 304.599,Z 920.9,A -85,B 0,C 180,E1 -15920.705,E2 -15920.705} C_VEL
LIN {X 0,Y 304.061,Z 926.085,A -85,B 0,C 180,E1 -15922.696,E2 -15922.696} C_VEL
LIN {X 0,Y 303.744,Z 929.894,A -85,B 0,C 180,E1 -15924.69,E2 -15924.69} C_VEL
LIN {X 0,Y 303.678,Z 931.646,A -85,B 0,C 180,E1 -15926.019,E2 -15926.019} C_VEL
LIN {X 0,Y 303.617,Z 932.901,A -85,B 0,C 180,E1 -15927.347,E2 -15927.347} C_VEL
LIN {X 0,Y 303.574,Z 933.68,A -85,B 0,C 180,E1 -15928.673,E2 -15928.673} C_VEL
LIN {X 0,Y 303.603,Z 933.975,A -85,B 0,C 180,E1 -15930,E2 -15930} C_VEL
LIN {X 0,Y 303.574,Z 933.675,A -85,B 0,C 180,E1 -15931.327,E2 -15931.327} C_VEL
LIN {X 0,Y 303.617,Z 932.887,A -85,B 0,C 180,E1 -15932.653,E2 -15932.653} C_VEL
LIN {X 0,Y 303.678,Z 931.623,A -85,B 0,C 180,E1 -15933.981,E2 -15933.981} C_VEL
LIN {X 0,Y 303.808,Z 928.847,A -85,B 0,C 180,E1 -15935.892,E2 -15935.892} C_VEL
LIN {X 0,Y 304.061,Z 926.044,A -85,B 0,C 180,E1 -15937.304,E2 -15937.304} C_VEL
LIN {X 0,Y 304.597,Z 920.845,A -85,B 0,C 180,E1 -15939.295,E2 -15939.295} C_VEL
LIN {X 0,Y 305.438,Z 913.997,A -85,B 0,C 180,E1 -15941.279,E2 -15941.279} C_VEL
LIN {X 0,Y 306.397,Z 906.517,A -85,B 0,C 180,E1 -15942.923,E2 -15942.923} C_VEL
LIN {X 0,Y 307.323,Z 899.142,A -85,B 0,C 180,E1 -15944.231,E2 -15944.231} C_VEL
LIN {X 0,Y 308.339,Z 891.248,A -85,B 0,C 180,E1 -15945.365,E2 -15945.365} C_VEL
LIN {X 0,Y 309.317,Z 882.906,A -85,B 0,C 180,E1 -15946.33,E2 -15946.33} C_VEL
LIN {X 0,Y 310.213,Z 872.241,A -85,B 0,C 180,E1 -15947.299,E2 -15947.299} C_VEL
LIN {X 0,Y 311.094,Z 860.623,A -85,B 0,C 180,E1 -15948.012,E2 -15948.012} C_VEL
LIN {X 0,Y 311.604,Z 850.871,A -85,B 0,C 180,E1 -15948.407,E2 -15948.407} C_VEL
LIN {X 0,Y 312.22,Z 807.631,A -85,B 0,C 180,E1 -15949.438,E2 -15949.438} C_VEL
LIN {X 0,Y 308.925,Z 784.523,A -85,B 0,C 180,E1 -15950.21,E2 -15950.21} C_VEL
LIN {X 0,Y 307.202,Z 774.221,A -85,B 0,C 180,E1 -15950.604,E2 -15950.604} C_VEL
LIN {X 0,Y 307.243,Z 773.093,A -85,B 0,C 180,E1 -15950.836,E2 -15950.836} C_VEL
LIN {X 0,Y 308.252,Z 764.923,A -85,B 0,C 180,E1 -15953.476,E2 -15953.476} C_VEL
LIN {X 0,Y 307.528,Z 759.474,A -85,B 0,C 180,E1 -15955.372,E2 -15955.372} C_VEL
LIN {X 0,Y 305.551,Z 749.348,A -85,B 0,C 180,E1 -15959.069,E2 -15959.069} C_VEL
LIN {X 0,Y 305.466,Z 749.251,A -85,B 0,C 180,E1 -15963.517,E2 -15963.517} C_VEL
LIN {X 0,Y 305.496,Z 749.235,A -85,B 0,C 180,E1 -15966.736,E2 -15966.736} C_VEL
LIN {X 0,Y 305.454,Z 749.228,A -85,B 0,C 180,E1 -15970.6,E2 -15970.6} C_VEL
LIN {X 0,Y 305.438,Z 749.244,A -85,B 0,C 180,E1 -15973.653,E2 -15973.653} C_VEL
LIN {X 0,Y 305.488,Z 749.227,A -85,B 0,C 180,E1 -15977.408,E2 -15977.408} C_VEL
LIN {X 0,Y 305.508,Z 749.186,A -85,B 0,C 180,E1 -15981.603,E2 -15981.603} C_VEL
LIN {X 0,Y 305.464,Z 749.24,A -85,B 0,C 180,E1 -15984.887,E2 -15984.887} C_VEL
LIN {X 0,Y 305.45,Z 749.243,A -85,B 0,C 180,E1 -15988.356,E2 -15988.356} C_VEL
LIN {X 0,Y 305.513,Z 749.223,A -85,B 0,C 180,E1 -15991.113,E2 -15991.113} C_VEL
LIN {X 0,Y 305.572,Z 749.236,A -85,B 0,C 180,E1 -15994.088,E2 -15994.088} C_VEL
LIN {X 0,Y 305.504,Z 749.219,A -85,B 0,C 180,E1 -15998.403,E2 -15998.403} C_VEL
LIN {X 0,Y 305.593,Z 749.225,A -85,B 0,C 180,E1 -16001.218,E2 -16001.218} C_VEL
LIN {X 0,Y 305.65,Z 749.216,A -85,B 0,C 180,E1 -16005.349,E2 -16005.349} C_VEL
LIN {X 0,Y 305.639,Z 749.21,A -85,B 0,C 180,E1 -16009.4,E2 -16009.4} C_VEL
LIN {X 0,Y 305.798,Z 749.205,A -85,B 0,C 180,E1 -16012.074,E2 -16012.074} C_VEL
LIN {X 0,Y 305.688,Z 749.21,A -85,B 0,C 180,E1 -16014.724,E2 -16014.724} C_VEL
LIN {X 0,Y 305.959,Z 749.16,A -85,B 0,C 180,E1 -16018.684,E2 -16018.684} C_VEL
LIN {X 0,Y 305.961,Z 749.182,A -85,B 0,C 180,E1 -16021.316,E2 -16021.316} C_VEL
LIN {X 0,Y 305.691,Z 749.206,A -85,B 0,C 180,E1 -16025.277,E2 -16025.277} C_VEL
LIN {X 0,Y 305.814,Z 749.173,A -85,B 0,C 180,E1 -16027.926,E2 -16027.926} C_VEL
LIN {X 0,Y 305.605,Z 749.227,A -85,B 0,C 180,E1 -16031.945,E2 -16031.945} C_VEL
LIN {X 0,Y 305.611,Z 749.217,A -85,B 0,C 180,E1 -16035.016,E2 -16035.016} C_VEL
LIN {X 0,Y 305.548,Z 749.229,A -85,B 0,C 180,E1 -16039.429,E2 -16039.429} C_VEL
LIN {X 0,Y 305.487,Z 749.241,A -85,B 0,C 180,E1 -16043.039,E2 -16043.039} C_VEL
LIN {X 0,Y 305.527,Z 749.217,A -85,B 0,C 180,E1 -16046.219,E2 -16046.219} C_VEL
LIN {X 0,Y 305.49,Z 749.243,A -85,B 0,C 180,E1 -16049.048,E2 -16049.048} C_VEL
LIN {X 0,Y 305.443,Z 749.241,A -85,B 0,C 180,E1 -16051.952,E2 -16051.952} C_VEL
LIN {X 0,Y 305.464,Z 749.24,A -85,B 0,C 180,E1 -16055.113,E2 -16055.113} C_VEL
LIN {X 0,Y 305.45,Z 749.245,A -85,B 0,C 180,E1 -16058.529,E2 -16058.529} C_VEL
LIN {X 0,Y 305.456,Z 749.193,A -85,B 0,C 180,E1 -16062.586,E2 -16062.586} C_VEL
LIN {X 0,Y 305.427,Z 749.249,A -85,B 0,C 180,E1 -16066.345,E2 -16066.345} C_VEL
LIN {X 0,Y 305.459,Z 749.233,A -85,B 0,C 180,E1 -16069.892,E2 -16069.892} C_VEL
LIN {X 0,Y 305.481,Z 749.236,A -85,B 0,C 180,E1 -16073.632,E2 -16073.632} C_VEL
LIN {X 0,Y 305.466,Z 749.245,A -85,B 0,C 180,E1 -16076.483,E2 -16076.483} C_VEL
LIN {X 0,Y 305.431,Z 749.242,A -85,B 0,C 180,E1 -16079.587,E2 -16079.587} C_VEL
LIN {X 0,Y 305.459,Z 749.247,A -85,B 0,C 180,E1 -16082.603,E2 -16082.603} C_VEL
LIN {X 0,Y 305.557,Z 749.467,A -85,B 0,C 180,E1 -16086.174,E2 -16086.174} C_VEL
LIN {X 0,Y 306.972,Z 757.335,A -85,B 0,C 180,E1 -16089.344,E2 -16089.344} C_VEL
LIN {X 0,Y 307.337,Z 758.921,A -85,B 0,C 180,E1 -16089.512,E2 -16089.512} C_VEL
LIN {X 0,Y 309.587,Z 767.227,A -85,B 0,C 180,E1 -16089.875,E2 -16089.875} C_VEL
LIN {X 0,Y 312.679,Z 783.524,A -85,B 0,C 180,E1 -16090.476,E2 -16090.476} C_VEL
LIN {X 0,Y 311.825,Z 833.386,A -85,B 0,C 180,E1 -16091.649,E2 -16091.649} C_VEL
LIN {X 0,Y 311.519,Z 843.148,A -85,B 0,C 180,E1 -16092.056,E2 -16092.056} C_VEL
LIN {X 0,Y 310.754,Z 854.223,A -85,B 0,C 180,E1 -16092.732,E2 -16092.732} C_VEL
LIN {X 0,Y 309.921,Z 865.021,A -85,B 0,C 180,E1 -16093.702,E2 -16093.702} C_VEL
LIN {X 0,Y 308.93,Z 873.407,A -85,B 0,C 180,E1 -16094.665,E2 -16094.665} C_VEL
LIN {X 0,Y 308.086,Z 881.317,A -85,B 0,C 180,E1 -16095.805,E2 -16095.805} C_VEL
LIN {X 0,Y 307.136,Z 888.694,A -85,B 0,C 180,E1 -16097.109,E2 -16097.109} C_VEL
LIN {X 0,Y 306.134,Z 896.163,A -85,B 0,C 180,E1 -16098.747,E2 -16098.747} C_VEL
LIN {X 0,Y 305.176,Z 903.01,A -85,B 0,C 180,E1 -16100.723,E2 -16100.723} C_VEL
LIN {X 0,Y 304.636,Z 907.762,A -85,B 0,C 180,E1 -16102.527,E2 -16102.527} C_VEL
LIN {X 0,Y 304.27,Z 910.83,A -85,B 0,C 180,E1 -16104.034,E2 -16104.034} C_VEL
LIN {X 0,Y 303.91,Z 913.735,A -85,B 0,C 180,E1 -16106.022,E2 -16106.022} C_VEL
LIN {X 0,Y 303.723,Z 915.003,A -85,B 0,C 180,E1 -16107.347,E2 -16107.347} C_VEL
LIN {X 0,Y 303.622,Z 915.803,A -85,B 0,C 180,E1 -16108.674,E2 -16108.674} C_VEL
LIN {X 0,Y 303.61,Z 916.107,A -85,B 0,C 180,E1 -16110,E2 -16110} C_VEL
LIN {X 0,Y 303.619,Z 915.83,A -85,B 0,C 180,E1 -16111.326,E2 -16111.326} C_VEL
LIN {X 0,Y 303.715,Z 915.083,A -85,B 0,C 180,E1 -16112.653,E2 -16112.653} C_VEL
LIN {X 0,Y 303.908,Z 913.867,A -85,B 0,C 180,E1 -16113.978,E2 -16113.978} C_VEL
LIN {X 0,Y 304.256,Z 911.018,A -85,B 0,C 180,E1 -16115.966,E2 -16115.966} C_VEL
LIN {X 0,Y 304.593,Z 908.01,A -85,B 0,C 180,E1 -16117.474,E2 -16117.474} C_VEL
LIN {X 0,Y 305.1,Z 903.324,A -85,B 0,C 180,E1 -16119.279,E2 -16119.279} C_VEL
LIN {X 0,Y 305.893,Z 897.829,A -85,B 0,C 180,E1 -16120.926,E2 -16120.926} C_VEL
LIN {X 0,Y 306.871,Z 890.922,A -85,B 0,C 180,E1 -16122.566,E2 -16122.566} C_VEL
LIN {X 0,Y 307.89,Z 882.989,A -85,B 0,C 180,E1 -16124.036,E2 -16124.036} C_VEL
LIN {X 0,Y 308.754,Z 875.424,A -85,B 0,C 180,E1 -16125.175,E2 -16125.175} C_VEL
LIN {X 0,Y 309.694,Z 867.488,A -85,B 0,C 180,E1 -16126.141,E2 -16126.141} C_VEL
LIN {X 0,Y 310.458,Z 859.288,A -85,B 0,C 180,E1 -16126.945,E2 -16126.945} C_VEL
LIN {X 0,Y 311.102,Z 850.97,A -85,B 0,C 180,E1 -16127.587,E2 -16127.587} C_VEL
LIN {X 0,Y 311.565,Z 841.97,A -85,B 0,C 180,E1 -16128.111,E2 -16128.111} C_VEL
LIN {X 0,Y 311.874,Z 832.561,A -85,B 0,C 180,E1 -16128.485,E2 -16128.485} C_VEL
LIN {X 0,Y 312.724,Z 783.645,A -85,B 0,C 180,E1 -16129.629,E2 -16129.629} C_VEL
LIN {X 0,Y 309.139,Z 765.183,A -85,B 0,C 180,E1 -16130.316,E2 -16130.316} C_VEL
LIN {X 0,Y 307.038,Z 757.765,A -85,B 0,C 180,E1 -16130.691,E2 -16130.691} C_VEL
LIN {X 0,Y 306.675,Z 755.363,A -85,B 0,C 180,E1 -16131.51,E2 -16131.51} C_VEL
LIN {X 0,Y 305.55,Z 749.337,A -85,B 0,C 180,E1 -16134.019,E2 -16134.019} C_VEL
LIN {X 0,Y 305.458,Z 749.247,A -85,B 0,C 180,E1 -16137.398,E2 -16137.398} C_VEL
LIN {X 0,Y 305.432,Z 749.244,A -85,B 0,C 180,E1 -16140.413,E2 -16140.413} C_VEL
LIN {X 0,Y 305.466,Z 749.247,A -85,B 0,C 180,E1 -16144.078,E2 -16144.078} C_VEL
LIN {X 0,Y 305.473,Z 749.235,A -85,B 0,C 180,E1 -16146.74,E2 -16146.74} C_VEL
LIN {X 0,Y 305.456,Z 749.237,A -85,B 0,C 180,E1 -16150.6,E2 -16150.6} C_VEL
LIN {X 0,Y 305.427,Z 749.249,A -85,B 0,C 180,E1 -16153.655,E2 -16153.655} C_VEL
LIN {X 0,Y 305.456,Z 749.194,A -85,B 0,C 180,E1 -16157.414,E2 -16157.414} C_VEL
LIN {X 0,Y 305.477,Z 749.241,A -85,B 0,C 180,E1 -16161.597,E2 -16161.597} C_VEL
LIN {X 0,Y 305.452,Z 749.238,A -85,B 0,C 180,E1 -16165.448,E2 -16165.448} C_VEL
LIN {X 0,Y 304.792,Z 749.318,A -85,B 0,C 180,E1 -16166.548,E2 -16166.548} C_VEL
LIN {X 0,Y 301.933,Z 749.68,A -85,B 0,C 180,E1 -16168.339,E2 -16168.339} C_VEL
LIN {X 0,Y 299.516,Z 749.987,A -85,B 0,C 180,E1 -16169.791,E2 -16169.791} C_VEL
LIN {X 0,Y 298.498,Z 750.116,A -85,B 0,C 180,E1 -16170.916,E2 -16170.916} C_VEL
LIN {X 0,Y 298.426,Z 750.119,A -85,B 0,C 180,E1 -16171.298,E2 -16171.298} C_VEL
LIN {X 0,Y 298.483,Z 750.096,A -85,B 0,C 180,E1 -16174.924,E2 -16174.924} C_VEL
LIN {X 0,Y 298.437,Z 750.12,A -85,B 0,C 180,E1 -16179.314,E2 -16179.314} C_VEL
LIN {X 0,Y 298.511,Z 750.091,A -85,B 0,C 180,E1 -16182.178,E2 -16182.178} C_VEL
LIN {X 0,Y 298.587,Z 750.091,A -85,B 0,C 180,E1 -16184.994,E2 -16184.994} C_VEL
LIN {X 0,Y 298.595,Z 750.099,A -85,B 0,C 180,E1 -16189.147,E2 -16189.147} C_VEL
LIN {X 0,Y 298.76,Z 750.052,A -85,B 0,C 180,E1 -16191.886,E2 -16191.886} C_VEL
LIN {X 0,Y 298.662,Z 750.081,A -85,B 0,C 180,E1 -16194.599,E2 -16194.599} C_VEL
LIN {X 0,Y 298.928,Z 750.057,A -85,B 0,C 180,E1 -16198.653,E2 -16198.653} C_VEL
LIN {X 0,Y 298.924,Z 750.036,A -85,B 0,C 180,E1 -16201.347,E2 -16201.347} C_VEL
LIN {X 0,Y 298.789,Z 750.076,A -85,B 0,C 180,E1 -16206.754,E2 -16206.754} C_VEL
LIN {X 0,Y 298.681,Z 750.085,A -85,B 0,C 180,E1 -16209.48,E2 -16209.48} C_VEL
LIN {X 0,Y 298.553,Z 750.087,A -85,B 0,C 180,E1 -16213.615,E2 -16213.615} C_VEL
LIN {X 0,Y 298.55,Z 750.108,A -85,B 0,C 180,E1 -16216.408,E2 -16216.408} C_VEL
LIN {X 0,Y 298.517,Z 750.099,A -85,B 0,C 180,E1 -16219.657,E2 -16219.657} C_VEL
LIN {X 0,Y 298.459,Z 750.111,A -85,B 0,C 180,E1 -16223.597,E2 -16223.597} C_VEL
LIN {X 0,Y 298.487,Z 750.113,A -85,B 0,C 180,E1 -16226.574,E2 -16226.574} C_VEL
LIN {X 0,Y 298.417,Z 750.105,A -85,B 0,C 180,E1 -16229.641,E2 -16229.641} C_VEL
LIN {X 0,Y 298.396,Z 750.128,A -85,B 0,C 180,E1 -16232.8,E2 -16232.8} C_VEL
LIN {X 0,Y 298.467,Z 750.092,A -85,B 0,C 180,E1 -16236.813,E2 -16236.813} C_VEL
LIN {X 0,Y 298.418,Z 750.081,A -85,B 0,C 180,E1 -16241.094,E2 -16241.094} C_VEL
LIN {X 0,Y 298.426,Z 750.116,A -85,B 0,C 180,E1 -16243.109,E2 -16243.109} C_VEL
LIN {X 0,Y 298.403,Z 750.114,A -85,B 0,C 180,E1 -16246.921,E2 -16246.921} C_VEL
LIN {X 0,Y 298.415,Z 750.124,A -85,B 0,C 180,E1 -16251.003,E2 -16251.003} C_VEL
LIN {X 0,Y 298.432,Z 750.11,A -85,B 0,C 180,E1 -16253.932,E2 -16253.932} C_VEL
LIN {X 0,Y 298.395,Z 750.105,A -85,B 0,C 180,E1 -16257.983,E2 -16257.983} C_VEL
LIN {X 0,Y 298.5,Z 750.332,A -85,B 0,C 180,E1 -16260.591,E2 -16260.591} C_VEL
LIN {X 0,Y 300.282,Z 759.311,A -85,B 0,C 180,E1 -16263.97,E2 -16263.97} C_VEL
LIN {X 0,Y 301.249,Z 765.241,A -85,B 0,C 180,E1 -16266.107,E2 -16266.107} C_VEL
LIN {X 0,Y 300.33,Z 773.51,A -85,B 0,C 180,E1 -16268.813,E2 -16268.813} C_VEL
LIN {X 0,Y 300.868,Z 777.038,A -85,B 0,C 180,E1 -16269.022,E2 -16269.022} C_VEL
LIN {X 0,Y 304.611,Z 800.988,A -85,B 0,C 180,E1 -16269.878,E2 -16269.878} C_VEL
LIN {X 0,Y 305.682,Z 810.903,A -85,B 0,C 180,E1 -16270.194,E2 -16270.194} C_VEL
LIN {X 0,Y 304.884,Z 851.271,A -85,B 0,C 180,E1 -16271.173,E2 -16271.173} C_VEL
LIN {X 0,Y 304.251,Z 862.463,A -85,B 0,C 180,E1 -16271.656,E2 -16271.656} C_VEL
LIN {X 0,Y 303.278,Z 874.17,A -85,B 0,C 180,E1 -16272.467,E2 -16272.467} C_VEL
LIN {X 0,Y 302.484,Z 882.87,A -85,B 0,C 180,E1 -16273.29,E2 -16273.29} C_VEL
LIN {X 0,Y 301.491,Z 891.179,A -85,B 0,C 180,E1 -16274.277,E2 -16274.277} C_VEL
LIN {X 0,Y 300.47,Z 899.045,A -85,B 0,C 180,E1 -16275.437,E2 -16275.437} C_VEL
LIN {X 0,Y 299.447,Z 906.403,A -85,B 0,C 180,E1 -16276.772,E2 -16276.772} C_VEL
LIN {X 0,Y 298.466,Z 913.872,A -85,B 0,C 180,E1 -16278.454,E2 -16278.454} C_VEL
LIN {X 0,Y 297.58,Z 920.692,A -85,B 0,C 180,E1 -16280.484,E2 -16280.484} C_VEL
LIN {X 0,Y 296.996,Z 925.877,A -85,B 0,C 180,E1 -16282.522,E2 -16282.522} C_VEL
LIN {X 0,Y 296.668,Z 929.685,A -85,B 0,C 180,E1 -16284.563,E2 -16284.563} C_VEL
LIN {X 0,Y 296.579,Z 931.438,A -85,B 0,C 180,E1 -16285.923,E2 -16285.923} C_VEL
LIN {X 0,Y 296.545,Z 932.693,A -85,B 0,C 180,E1 -16287.283,E2 -16287.283} C_VEL
LIN {X 0,Y 296.493,Z 933.471,A -85,B 0,C 180,E1 -16288.642,E2 -16288.642} C_VEL
LIN {X 0,Y 296.518,Z 933.767,A -85,B 0,C 180,E1 -16290,E2 -16290} C_VEL
LIN {X 0,Y 296.493,Z 933.467,A -85,B 0,C 180,E1 -16291.358,E2 -16291.358} C_VEL
LIN {X 0,Y 296.545,Z 932.678,A -85,B 0,C 180,E1 -16292.717,E2 -16292.717} C_VEL
LIN {X 0,Y 296.579,Z 931.413,A -85,B 0,C 180,E1 -16294.077,E2 -16294.077} C_VEL
LIN {X 0,Y 296.695,Z 929.031,A -85,B 0,C 180,E1 -16295.802,E2 -16295.802} C_VEL
LIN {X 0,Y 296.996,Z 925.833,A -85,B 0,C 180,E1 -16297.478,E2 -16297.478} C_VEL
LIN {X 0,Y 297.577,Z 920.634,A -85,B 0,C 180,E1 -16299.516,E2 -16299.516} C_VEL
LIN {X 0,Y 298.464,Z 913.786,A -85,B 0,C 180,E1 -16301.546,E2 -16301.546} C_VEL
LIN {X 0,Y 299.445,Z 906.305,A -85,B 0,C 180,E1 -16303.228,E2 -16303.228} C_VEL
LIN {X 0,Y 300.447,Z 898.931,A -85,B 0,C 180,E1 -16304.564,E2 -16304.564} C_VEL
LIN {X 0,Y 301.471,Z 891.035,A -85,B 0,C 180,E1 -16305.724,E2 -16305.724} C_VEL
LIN {X 0,Y 302.515,Z 882.693,A -85,B 0,C 180,E1 -16306.708,E2 -16306.708} C_VEL
LIN {X 0,Y 303.453,Z 872.027,A -85,B 0,C 180,E1 -16307.697,E2 -16307.697} C_VEL
LIN {X 0,Y 304.36,Z 860.405,A -85,B 0,C 180,E1 -16308.425,E2 -16308.425} C_VEL
LIN {X 0,Y 304.874,Z 850.647,A -85,B 0,C 180,E1 -16308.828,E2 -16308.828} C_VEL
LIN {X 0,Y 305.57,Z 808.769,A -85,B 0,C 180,E1 -16309.845,E2 -16309.845} C_VEL
LIN {X 0,Y 302.119,Z 784.633,A -85,B 0,C 180,E1 -16310.677,E2 -16310.677} C_VEL
LIN {X 0,Y 300.33,Z 773.939,A -85,B 0,C 180,E1 -16311.105,E2 -16311.105} C_VEL
LIN {X 0,Y 300.358,Z 772.883,A -85,B 0,C 180,E1 -16311.337,E2 -16311.337} C_VEL
LIN {X 0,Y 301.249,Z 765.192,A -85,B 0,C 180,E1 -16313.893,E2 -16313.893} C_VEL
LIN {X 0,Y 300.115,Z 758.186,A -85,B 0,C 180,E1 -16316.419,E2 -16316.419} C_VEL
LIN {X 0,Y 298.482,Z 750.141,A -85,B 0,C 180,E1 -16319.521,E2 -16319.521} C_VEL
LIN {X 0,Y 298.396,Z 750.123,A -85,B 0,C 180,E1 -16322.8,E2 -16322.8} C_VEL
LIN {X 0,Y 298.465,Z 750.111,A -85,B 0,C 180,E1 -16326.812,E2 -16326.812} C_VEL
LIN {X 0,Y 298.387,Z 750.105,A -85,B 0,C 180,E1 -16331.088,E2 -16331.088} C_VEL
LIN {X 0,Y 298.399,Z 750.116,A -85,B 0,C 180,E1 -16333.103,E2 -16333.103} C_VEL
LIN {X 0,Y 298.432,Z 750.113,A -85,B 0,C 180,E1 -16336.926,E2 -16336.926} C_VEL
LIN {X 0,Y 298.425,Z 750.062,A -85,B 0,C 180,E1 -16341.001,E2 -16341.001} C_VEL
LIN {X 0,Y 298.433,Z 750.104,A -85,B 0,C 180,E1 -16343.932,E2 -16343.932} C_VEL
LIN {X 0,Y 298.395,Z 750.125,A -85,B 0,C 180,E1 -16347.984,E2 -16347.984} C_VEL
LIN {X 0,Y 298.459,Z 750.107,A -85,B 0,C 180,E1 -16351.904,E2 -16351.904} C_VEL
LIN {X 0,Y 298.487,Z 750.114,A -85,B 0,C 180,E1 -16354.924,E2 -16354.924} C_VEL
LIN {X 0,Y 298.454,Z 750.099,A -85,B 0,C 180,E1 -16359.316,E2 -16359.316} C_VEL
LIN {X 0,Y 298.54,Z 750.109,A -85,B 0,C 180,E1 -16362.18,E2 -16362.18} C_VEL
LIN {X 0,Y 298.595,Z 750.095,A -85,B 0,C 180,E1 -16364.995,E2 -16364.995} C_VEL
LIN {X 0,Y 298.594,Z 750.086,A -85,B 0,C 180,E1 -16369.147,E2 -16369.147} C_VEL
LIN {X 0,Y 298.746,Z 750.082,A -85,B 0,C 180,E1 -16371.886,E2 -16371.886} C_VEL
LIN {X 0,Y 298.659,Z 750.087,A -85,B 0,C 180,E1 -16374.599,E2 -16374.599} C_VEL
LIN {X 0,Y 298.925,Z 750.035,A -85,B 0,C 180,E1 -16378.653,E2 -16378.653} C_VEL
LIN {X 0,Y 298.928,Z 750.058,A -85,B 0,C 180,E1 -16381.347,E2 -16381.347} C_VEL
LIN {X 0,Y 298.662,Z 750.081,A -85,B 0,C 180,E1 -16385.401,E2 -16385.401} C_VEL
LIN {X 0,Y 298.76,Z 750.052,A -85,B 0,C 180,E1 -16388.114,E2 -16388.114} C_VEL
LIN {X 0,Y 298.555,Z 750.107,A -85,B 0,C 180,E1 -16392.232,E2 -16392.232} C_VEL
LIN {X 0,Y 298.551,Z 750.095,A -85,B 0,C 180,E1 -16395.169,E2 -16395.169} C_VEL
LIN {X 0,Y 298.509,Z 750.102,A -85,B 0,C 180,E1 -16399.245,E2 -16399.245} C_VEL
LIN {X 0,Y 298.43,Z 750.115,A -85,B 0,C 180,E1 -16403.6,E2 -16403.6} C_VEL
LIN {X 0,Y 298.486,Z 750.095,A -85,B 0,C 180,E1 -16406.575,E2 -16406.575} C_VEL
LIN {X 0,Y 298.418,Z 750.125,A -85,B 0,C 180,E1 -16409.641,E2 -16409.641} C_VEL
LIN {X 0,Y 298.396,Z 750.114,A -85,B 0,C 180,E1 -16412.8,E2 -16412.8} C_VEL
LIN {X 0,Y 298.448,Z 750.121,A -85,B 0,C 180,E1 -16416.808,E2 -16416.808} C_VEL
LIN {X 0,Y 298.387,Z 750.085,A -85,B 0,C 180,E1 -16421.088,E2 -16421.088} C_VEL
LIN {X 0,Y 298.4,Z 750.073,A -85,B 0,C 180,E1 -16423.103,E2 -16423.103} C_VEL
LIN {X 0,Y 298.404,Z 750.125,A -85,B 0,C 180,E1 -16426.921,E2 -16426.921} C_VEL
LIN {X 0,Y 298.4,Z 750.1,A -85,B 0,C 180,E1 -16431.008,E2 -16431.008} C_VEL
LIN {X 0,Y 298.419,Z 750.119,A -85,B 0,C 180,E1 -16433.93,E2 -16433.93} C_VEL
LIN {X 0,Y 298.394,Z 750.116,A -85,B 0,C 180,E1 -16437.2,E2 -16437.2} C_VEL
LIN {X 0,Y 298.403,Z 750.127,A -85,B 0,C 180,E1 -16440.625,E2 -16440.625} C_VEL
LIN {X 0,Y 298.451,Z 750.122,A -85,B 0,C 180,E1 -16444.921,E2 -16444.921} C_VEL
LIN {X 0,Y 298.512,Z 750.347,A -85,B 0,C 180,E1 -16445.854,E2 -16445.854} C_VEL
LIN {X 0,Y 299.849,Z 757.608,A -85,B 0,C 180,E1 -16448.843,E2 -16448.843} C_VEL
LIN {X 0,Y 300.383,Z 759.498,A -85,B 0,C 180,E1 -16449.029,E2 -16449.029} C_VEL
LIN {X 0,Y 302.958,Z 768.365,A -85,B 0,C 180,E1 -16449.438,E2 -16449.438} C_VEL
LIN {X 0,Y 306.06,Z 785.214,A -85,B 0,C 180,E1 -16450.071,E2 -16450.071} C_VEL
LIN {X 0,Y 305.112,Z 833.612,A -85,B 0,C 180,E1 -16451.231,E2 -16451.231} C_VEL
LIN {X 0,Y 304.789,Z 843.368,A -85,B 0,C 180,E1 -16451.646,E2 -16451.646} C_VEL
LIN {X 0,Y 303.989,Z 854.439,A -85,B 0,C 180,E1 -16452.336,E2 -16452.336} C_VEL
LIN {X 0,Y 303.13,Z 865.235,A -85,B 0,C 180,E1 -16453.327,E2 -16453.327} C_VEL
LIN {X 0,Y 302.116,Z 873.619,A -85,B 0,C 180,E1 -16454.31,E2 -16454.31} C_VEL
LIN {X 0,Y 301.219,Z 881.529,A -85,B 0,C 180,E1 -16455.474,E2 -16455.474} C_VEL
LIN {X 0,Y 300.473,Z 887.209,A -85,B 0,C 180,E1 -16456.473,E2 -16456.473} C_VEL
LIN {X 0,Y 299.577,Z 893.551,A -85,B 0,C 180,E1 -16457.811,E2 -16457.811} C_VEL
LIN {X 0,Y 298.777,Z 898.823,A -85,B 0,C 180,E1 -16459.153,E2 -16459.153} C_VEL
LIN {X 0,Y 298.165,Z 903.221,A -85,B 0,C 180,E1 -16460.503,E2 -16460.503} C_VEL
LIN {X 0,Y 297.76,Z 906.879,A -85,B 0,C 180,E1 -16461.859,E2 -16461.859} C_VEL
LIN {X 0,Y 297.228,Z 910.663,A -85,B 0,C 180,E1 -16463.667,E2 -16463.667} C_VEL
LIN {X 0,Y 297.085,Z 912.184,A -85,B 0,C 180,E1 -16464.57,E2 -16464.57} C_VEL
LIN {X 0,Y 296.853,Z 913.943,A -85,B 0,C 180,E1 -16465.927,E2 -16465.927} C_VEL
LIN {X 0,Y 296.652,Z 915.212,A -85,B 0,C 180,E1 -16467.284,E2 -16467.284} C_VEL
LIN {X 0,Y 296.541,Z 916.012,A -85,B 0,C 180,E1 -16468.642,E2 -16468.642} C_VEL
LIN {X 0,Y 296.526,Z 916.316,A -85,B 0,C 180,E1 -16470,E2 -16470} C_VEL
LIN {X 0,Y 296.538,Z 916.038,A -85,B 0,C 180,E1 -16471.358,E2 -16471.358} C_VEL
LIN {X 0,Y 296.644,Z 915.29,A -85,B 0,C 180,E1 -16472.716,E2 -16472.716} C_VEL
LIN {X 0,Y 296.85,Z 914.074,A -85,B 0,C 180,E1 -16474.073,E2 -16474.073} C_VEL
LIN {X 0,Y 297.077,Z 912.37,A -85,B 0,C 180,E1 -16475.43,E2 -16475.43} C_VEL
LIN {X 0,Y 297.497,Z 908.784,A -85,B 0,C 180,E1 -16477.397,E2 -16477.397} C_VEL
LIN {X 0,Y 298.1,Z 903.531,A -85,B 0,C 180,E1 -16479.499,E2 -16479.499} C_VEL
LIN {X 0,Y 298.947,Z 898.036,A -85,B 0,C 180,E1 -16481.183,E2 -16481.183} C_VEL
LIN {X 0,Y 299.965,Z 891.128,A -85,B 0,C 180,E1 -16482.861,E2 -16482.861} C_VEL
LIN {X 0,Y 301.023,Z 883.194,A -85,B 0,C 180,E1 -16484.363,E2 -16484.363} C_VEL
LIN {X 0,Y 301.908,Z 875.629,A -85,B 0,C 180,E1 -16485.528,E2 -16485.528} C_VEL
LIN {X 0,Y 302.881,Z 867.691,A -85,B 0,C 180,E1 -16486.514,E2 -16486.514} C_VEL
LIN {X 0,Y 303.693,Z 859.49,A -85,B 0,C 180,E1 -16487.335,E2 -16487.335} C_VEL
LIN {X 0,Y 304.366,Z 851.17,A -85,B 0,C 180,E1 -16487.989,E2 -16487.989} C_VEL
LIN {X 0,Y 304.838,Z 842.167,A -85,B 0,C 180,E1 -16488.525,E2 -16488.525} C_VEL
LIN {X 0,Y 305.158,Z 833.04,A -85,B 0,C 180,E1 -16488.897,E2 -16488.897} C_VEL
LIN {X 0,Y 305.992,Z 784.169,A -85,B 0,C 180,E1 -16490.071,E2 -16490.071} C_VEL
LIN {X 0,Y 302.362,Z 765.823,A -85,B 0,C 180,E1 -16490.781,E2 -16490.781} C_VEL
LIN {X 0,Y 299.972,Z 758.102,A -85,B 0,C 180,E1 -16491.186,E2 -16491.186} C_VEL
LIN {X 0,Y 299.748,Z 756.941,A -85,B 0,C 180,E1 -16491.491,E2 -16491.491} C_VEL
LIN {X 0,Y 298.514,Z 750.202,A -85,B 0,C 180,E1 -16494.377,E2 -16494.377} C_VEL
LIN {X 0,Y 298.415,Z 750.122,A -85,B 0,C 180,E1 -16498.101,E2 -16498.101} C_VEL
LIN {X 0,Y 298.389,Z 750.11,A -85,B 0,C 180,E1 -16502.014,E2 -16502.014} C_VEL
LIN {X 0,Y 298.419,Z 750.122,A -85,B 0,C 180,E1 -16506.07,E2 -16506.07} C_VEL
LIN {X 0,Y 298.402,Z 750.103,A -85,B 0,C 180,E1 -16509.487,E2 -16509.487} C_VEL
LIN {X 0,Y 298.4,Z 750.126,A -85,B 0,C 180,E1 -16513.103,E2 -16513.103} C_VEL
LIN {X 0,Y 298.404,Z 750.074,A -85,B 0,C 180,E1 -16516.921,E2 -16516.921} C_VEL
LIN {X 0,Y 298.405,Z 750.114,A -85,B 0,C 180,E1 -16521.006,E2 -16521.006} C_VEL
LIN {X 0,Y 298.42,Z 750.123,A -85,B 0,C 180,E1 -16523.93,E2 -16523.93} C_VEL
LIN {X 0,Y 298.395,Z 750.118,A -85,B 0,C 180,E1 -16527.984,E2 -16527.984} C_VEL
LIN {X 0,Y 298.426,Z 750.119,A -85,B 0,C 180,E1 -16531.298,E2 -16531.298} C_VEL
LIN {X 0,Y 297.778,Z 750.197,A -85,B 0,C 180,E1 -16532.423,E2 -16532.423} C_VEL
LIN {X 0,Y 294.91,Z 750.546,A -85,B 0,C 180,E1 -16534.256,E2 -16534.256} C_VEL
LIN {X 0,Y 292.475,Z 750.854,A -85,B 0,C 180,E1 -16535.743,E2 -16535.743} C_VEL
LIN {X 0,Y 291.448,Z 750.988,A -85,B 0,C 180,E1 -16536.896,E2 -16536.896} C_VEL
LIN {X 0,Y 291.375,Z 751.001,A -85,B 0,C 180,E1 -16537.287,E2 -16537.287} C_VEL
LIN {X 0,Y 291.459,Z 750.986,A -85,B 0,C 180,E1 -16540.27,E2 -16540.27} C_VEL
LIN {X 0,Y 291.516,Z 750.97,A -85,B 0,C 180,E1 -16544.653,E2 -16544.653} C_VEL
LIN {X 0,Y 291.539,Z 750.981,A -85,B 0,C 180,E1 -16548.881,E2 -16548.881} C_VEL
LIN {X 0,Y 291.71,Z 750.931,A -85,B 0,C 180,E1 -16551.688,E2 -16551.688} C_VEL
LIN {X 0,Y 291.633,Z 750.956,A -85,B 0,C 180,E1 -16554.468,E2 -16554.468} C_VEL
LIN {X 0,Y 291.894,Z 750.934,A -85,B 0,C 180,E1 -16558.62,E2 -16558.62} C_VEL
LIN {X 0,Y 291.89,Z 750.911,A -85,B 0,C 180,E1 -16561.38,E2 -16561.38} C_VEL
LIN {X 0,Y 291.738,Z 750.955,A -85,B 0,C 180,E1 -16566.918,E2 -16566.918} C_VEL
LIN {X 0,Y 291.63,Z 750.96,A -85,B 0,C 180,E1 -16569.712,E2 -16569.712} C_VEL
LIN {X 0,Y 291.523,Z 750.966,A -85,B 0,C 180,E1 -16573.95,E2 -16573.95} C_VEL
LIN {X 0,Y 291.489,Z 750.986,A -85,B 0,C 180,E1 -16576.818,E2 -16576.818} C_VEL
LIN {X 0,Y 291.452,Z 750.975,A -85,B 0,C 180,E1 -16579.875,E2 -16579.875} C_VEL
LIN {X 0,Y 291.402,Z 750.996,A -85,B 0,C 180,E1 -16584.205,E2 -16584.205} C_VEL
LIN {X 0,Y 291.42,Z 750.992,A -85,B 0,C 180,E1 -16587.272,E2 -16587.272} C_VEL
LIN {X 0,Y 291.335,Z 750.992,A -85,B 0,C 180,E1 -16590.437,E2 -16590.437} C_VEL
LIN {X 0,Y 291.345,Z 751.006,A -85,B 0,C 180,E1 -16593.698,E2 -16593.698} C_VEL
LIN {X 0,Y 291.399,Z 750.959,A -85,B 0,C 180,E1 -16597.26,E2 -16597.26} C_VEL
LIN {X 0,Y 291.376,Z 750.949,A -85,B 0,C 180,E1 -16600.635,E2 -16600.635} C_VEL
LIN {X 0,Y 291.302,Z 751.012,A -85,B 0,C 180,E1 -16604.399,E2 -16604.399} C_VEL
LIN {X 0,Y 291.326,Z 750.983,A -85,B 0,C 180,E1 -16608.404,E2 -16608.404} C_VEL
LIN {X 0,Y 291.365,Z 751.004,A -85,B 0,C 180,E1 -16611.16,E2 -16611.16} C_VEL
LIN {X 0,Y 291.385,Z 750.989,A -85,B 0,C 180,E1 -16614.629,E2 -16614.629} C_VEL
LIN {X 0,Y 291.372,Z 750.979,A -85,B 0,C 180,E1 -16617.951,E2 -16617.951} C_VEL
LIN {X 0,Y 291.413,Z 751.025,A -85,B 0,C 180,E1 -16620.073,E2 -16620.073} C_VEL
LIN {X 0,Y 293.03,Z 759.108,A -85,B 0,C 180,E1 -16623.276,E2 -16623.276} C_VEL
LIN {X 0,Y 294.257,Z 766.562,A -85,B 0,C 180,E1 -16626.045,E2 -16626.045} C_VEL
LIN {X 0,Y 293.483,Z 773.353,A -85,B 0,C 180,E1 -16628.303,E2 -16628.303} C_VEL
LIN {X 0,Y 294.135,Z 777.557,A -85,B 0,C 180,E1 -16628.536,E2 -16628.536} C_VEL
LIN {X 0,Y 297.971,Z 801.969,A -85,B 0,C 180,E1 -16629.439,E2 -16629.439} C_VEL
LIN {X 0,Y 299.007,Z 810.609,A -85,B 0,C 180,E1 -16629.73,E2 -16629.73} C_VEL
LIN {X 0,Y 298.189,Z 849.974,A -85,B 0,C 180,E1 -16630.695,E2 -16630.695} C_VEL
LIN {X 0,Y 297.738,Z 858.939,A -85,B 0,C 180,E1 -16631.061,E2 -16631.061} C_VEL
LIN {X 0,Y 297.019,Z 868.573,A -85,B 0,C 180,E1 -16631.639,E2 -16631.639} C_VEL
LIN {X 0,Y 296.22,Z 877.72,A -85,B 0,C 180,E1 -16632.392,E2 -16632.392} C_VEL
LIN {X 0,Y 294.994,Z 888.509,A -85,B 0,C 180,E1 -16633.566,E2 -16633.566} C_VEL
LIN {X 0,Y 293.896,Z 896.793,A -85,B 0,C 180,E1 -16634.749,E2 -16634.749} C_VEL
LIN {X 0,Y 292.761,Z 904.487,A -85,B 0,C 180,E1 -16636.11,E2 -16636.11} C_VEL
LIN {X 0,Y 291.903,Z 910.824,A -85,B 0,C 180,E1 -16637.485,E2 -16637.485} C_VEL
LIN {X 0,Y 291.157,Z 916.091,A -85,B 0,C 180,E1 -16638.866,E2 -16638.866} C_VEL
LIN {X 0,Y 290.57,Z 920.484,A -85,B 0,C 180,E1 -16640.252,E2 -16640.252} C_VEL
LIN {X 0,Y 289.927,Z 925.668,A -85,B 0,C 180,E1 -16642.338,E2 -16642.338} C_VEL
LIN {X 0,Y 289.603,Z 929.478,A -85,B 0,C 180,E1 -16644.429,E2 -16644.429} C_VEL
LIN {X 0,Y 289.484,Z 931.229,A -85,B 0,C 180,E1 -16645.823,E2 -16645.823} C_VEL
LIN {X 0,Y 289.451,Z 932.484,A -85,B 0,C 180,E1 -16647.217,E2 -16647.217} C_VEL
LIN {X 0,Y 289.415,Z 933.263,A -85,B 0,C 180,E1 -16648.609,E2 -16648.609} C_VEL
LIN {X 0,Y 289.435,Z 933.558,A -85,B 0,C 180,E1 -16650,E2 -16650} C_VEL
LIN {X 0,Y 289.415,Z 933.258,A -85,B 0,C 180,E1 -16651.391,E2 -16651.391} C_VEL
LIN {X 0,Y 289.451,Z 932.469,A -85,B 0,C 180,E1 -16652.783,E2 -16652.783} C_VEL
LIN {X 0,Y 289.484,Z 931.204,A -85,B 0,C 180,E1 -16654.177,E2 -16654.177} C_VEL
LIN {X 0,Y 289.684,Z 928.284,A -85,B 0,C 180,E1 -16656.267,E2 -16656.267} C_VEL
LIN {X 0,Y 289.927,Z 925.622,A -85,B 0,C 180,E1 -16657.662,E2 -16657.662} C_VEL
LIN {X 0,Y 290.567,Z 920.423,A -85,B 0,C 180,E1 -16659.748,E2 -16659.748} C_VEL
LIN {X 0,Y 291.485,Z 913.574,A -85,B 0,C 180,E1 -16661.826,E2 -16661.826} C_VEL
LIN {X 0,Y 292.519,Z 906.093,A -85,B 0,C 180,E1 -16663.548,E2 -16663.548} C_VEL
LIN {X 0,Y 293.583,Z 898.719,A -85,B 0,C 180,E1 -16664.912,E2 -16664.912} C_VEL
LIN {X 0,Y 294.648,Z 890.823,A -85,B 0,C 180,E1 -16666.098,E2 -16666.098} C_VEL
LIN {X 0,Y 295.721,Z 882.48,A -85,B 0,C 180,E1 -16667.104,E2 -16667.104} C_VEL
LIN {X 0,Y 296.666,Z 871.811,A -85,B 0,C 180,E1 -16668.115,E2 -16668.115} C_VEL
LIN {X 0,Y 297.634,Z 860.186,A -85,B 0,C 180,E1 -16668.857,E2 -16668.857} C_VEL
LIN {X 0,Y 298.148,Z 850.422,A -85,B 0,C 180,E1 -16669.269,E2 -16669.269} C_VEL
LIN {X 0,Y 298.911,Z 809.551,A -85,B 0,C 180,E1 -16670.281,E2 -16670.281} C_VEL
LIN {X 0,Y 295.656,Z 786.684,A -85,B 0,C 180,E1 -16671.092,E2 -16671.092} C_VEL
LIN {X 0,Y 293.471,Z 773.742,A -85,B 0,C 180,E1 -16671.62,E2 -16671.62} C_VEL
LIN {X 0,Y 293.483,Z 772.672,A -85,B 0,C 180,E1 -16671.862,E2 -16671.862} C_VEL
LIN {X 0,Y 294.256,Z 766.512,A -85,B 0,C 180,E1 -16673.956,E2 -16673.956} C_VEL
LIN {X 0,Y 293.034,Z 759.048,A -85,B 0,C 180,E1 -16676.724,E2 -16676.724} C_VEL
LIN {X 0,Y 291.431,Z 751.02,A -85,B 0,C 180,E1 -16679.898,E2 -16679.898} C_VEL
LIN {X 0,Y 291.345,Z 751.01,A -85,B 0,C 180,E1 -16683.698,E2 -16683.698} C_VEL
LIN {X 0,Y 291.394,Z 750.995,A -85,B 0,C 180,E1 -16687.259,E2 -16687.259} C_VEL
LIN {X 0,Y 291.334,Z 750.985,A -85,B 0,C 180,E1 -16690.642,E2 -16690.642} C_VEL
LIN {X 0,Y 291.294,Z 751.011,A -85,B 0,C 180,E1 -16694.401,E2 -16694.401} C_VEL
LIN {X 0,Y 291.356,Z 750.969,A -85,B 0,C 180,E1 -16698.398,E2 -16698.398} C_VEL
LIN {X 0,Y 291.374,Z 750.94,A -85,B 0,C 180,E1 -16701.162,E2 -16701.162} C_VEL
LIN {X 0,Y 291.386,Z 750.993,A -85,B 0,C 180,E1 -16704.63,E2 -16704.63} C_VEL
LIN {X 0,Y 291.371,Z 751,A -85,B 0,C 180,E1 -16707.951,E2 -16707.951} C_VEL
LIN {X 0,Y 291.378,Z 750.984,A -85,B 0,C 180,E1 -16711.158,E2 -16711.158} C_VEL
LIN {X 0,Y 291.416,Z 750.998,A -85,B 0,C 180,E1 -16714.272,E2 -16714.272} C_VEL
LIN {X 0,Y 291.384,Z 750.986,A -85,B 0,C 180,E1 -16717.3,E2 -16717.3} C_VEL
LIN {X 0,Y 291.461,Z 750.977,A -85,B 0,C 180,E1 -16720.271,E2 -16720.271} C_VEL
LIN {X 0,Y 291.556,Z 750.973,A -85,B 0,C 180,E1 -16724.624,E2 -16724.624} C_VEL
LIN {X 0,Y 291.538,Z 750.96,A -85,B 0,C 180,E1 -16728.881,E2 -16728.881} C_VEL
LIN {X 0,Y 291.699,Z 750.959,A -85,B 0,C 180,E1 -16731.688,E2 -16731.688} C_VEL
LIN {X 0,Y 291.629,Z 750.964,A -85,B 0,C 180,E1 -16734.468,E2 -16734.468} C_VEL
LIN {X 0,Y 291.891,Z 750.91,A -85,B 0,C 180,E1 -16738.62,E2 -16738.62} C_VEL
LIN {X 0,Y 291.894,Z 750.934,A -85,B 0,C 180,E1 -16741.38,E2 -16741.38} C_VEL
LIN {X 0,Y 291.748,Z 750.925,A -85,B 0,C 180,E1 -16746.918,E2 -16746.918} C_VEL
LIN {X 0,Y 291.631,Z 750.958,A -85,B 0,C 180,E1 -16749.712,E2 -16749.712} C_VEL
LIN {X 0,Y 291.517,Z 750.981,A -85,B 0,C 180,E1 -16753.951,E2 -16753.951} C_VEL
LIN {X 0,Y 291.444,Z 750.968,A -85,B 0,C 180,E1 -16756.821,E2 -16756.821} C_VEL
LIN {X 0,Y 291.425,Z 750.99,A -85,B 0,C 180,E1 -16759.86,E2 -16759.86} C_VEL
LIN {X 0,Y 291.384,Z 750.992,A -85,B 0,C 180,E1 -16764.207,E2 -16764.207} C_VEL
LIN {X 0,Y 291.42,Z 750.981,A -85,B 0,C 180,E1 -16767.272,E2 -16767.272} C_VEL
LIN {X 0,Y 291.336,Z 751.006,A -85,B 0,C 180,E1 -16770.437,E2 -16770.437} C_VEL
LIN {X 0,Y 291.346,Z 750.989,A -85,B 0,C 180,E1 -16773.698,E2 -16773.698} C_VEL
LIN {X 0,Y 291.378,Z 751.003,A -85,B 0,C 180,E1 -16777.254,E2 -16777.254} C_VEL
LIN {X 0,Y 291.333,Z 750.97,A -85,B 0,C 180,E1 -16780.643,E2 -16780.643} C_VEL
LIN {X 0,Y 291.29,Z 750.976,A -85,B 0,C 180,E1 -16784.402,E2 -16784.402} C_VEL
LIN {X 0,Y 291.328,Z 751.007,A -85,B 0,C 180,E1 -16788.404,E2 -16788.404} C_VEL
LIN {X 0,Y 291.348,Z 750.977,A -85,B 0,C 180,E1 -16791.158,E2 -16791.158} C_VEL
LIN {X 0,Y 291.362,Z 751.006,A -85,B 0,C 180,E1 -16794.626,E2 -16794.626} C_VEL
LIN {X 0,Y 291.367,Z 750.985,A -85,B 0,C 180,E1 -16797.95,E2 -16797.95} C_VEL
LIN {X 0,Y 291.346,Z 751.007,A -85,B 0,C 180,E1 -16801.154,E2 -16801.154} C_VEL
LIN {X 0,Y 291.459,Z 751.149,A -85,B 0,C 180,E1 -16805.468,E2 -16805.468} C_VEL
LIN {X 0,Y 292.719,Z 757.805,A -85,B 0,C 180,E1 -16808.298,E2 -16808.298} C_VEL
LIN {X 0,Y 293.264,Z 759.712,A -85,B 0,C 180,E1 -16808.494,E2 -16808.494} C_VEL
LIN {X 0,Y 296.163,Z 768.888,A -85,B 0,C 180,E1 -16808.951,E2 -16808.951} C_VEL
LIN {X 0,Y 299.392,Z 786.361,A -85,B 0,C 180,E1 -16809.631,E2 -16809.631} C_VEL
LIN {X 0,Y 298.419,Z 833.838,A -85,B 0,C 180,E1 -16810.793,E2 -16810.793} C_VEL
LIN {X 0,Y 298.08,Z 843.587,A -85,B 0,C 180,E1 -16811.217,E2 -16811.217} C_VEL
LIN {X 0,Y 297.244,Z 854.655,A -85,B 0,C 180,E1 -16811.921,E2 -16811.921} C_VEL
LIN {X 0,Y 296.353,Z 865.448,A -85,B 0,C 180,E1 -16812.934,E2 -16812.934} C_VEL
LIN {X 0,Y 295.287,Z 873.832,A -85,B 0,C 180,E1 -16813.938,E2 -16813.938} C_VEL
LIN {X 0,Y 294.363,Z 881.741,A -85,B 0,C 180,E1 -16815.128,E2 -16815.128} C_VEL
LIN {X 0,Y 293.322,Z 889.117,A -85,B 0,C 180,E1 -16816.49,E2 -16816.49} C_VEL
LIN {X 0,Y 292.224,Z 896.586,A -85,B 0,C 180,E1 -16818.204,E2 -16818.204} C_VEL
LIN {X 0,Y 291.173,Z 903.431,A -85,B 0,C 180,E1 -16820.273,E2 -16820.273} C_VEL
LIN {X 0,Y 290.489,Z 908.599,A -85,B 0,C 180,E1 -16822.353,E2 -16822.353} C_VEL
LIN {X 0,Y 290.121,Z 911.228,A -85,B 0,C 180,E1 -16823.728,E2 -16823.728} C_VEL
LIN {X 0,Y 289.775,Z 914.153,A -85,B 0,C 180,E1 -16825.827,E2 -16825.827} C_VEL
LIN {X 0,Y 289.583,Z 915.421,A -85,B 0,C 180,E1 -16827.218,E2 -16827.218} C_VEL
LIN {X 0,Y 289.462,Z 916.22,A -85,B 0,C 180,E1 -16828.609,E2 -16828.609} C_VEL
LIN {X 0,Y 289.443,Z 916.524,A -85,B 0,C 180,E1 -16830,E2 -16830} C_VEL
LIN {X 0,Y 289.46,Z 916.246,A -85,B 0,C 180,E1 -16831.391,E2 -16831.391} C_VEL
LIN {X 0,Y 289.576,Z 915.498,A -85,B 0,C 180,E1 -16832.782,E2 -16832.782} C_VEL
LIN {X 0,Y 289.773,Z 914.283,A -85,B 0,C 180,E1 -16834.173,E2 -16834.173} C_VEL
LIN {X 0,Y 290.11,Z 911.445,A -85,B 0,C 180,E1 -16836.252,E2 -16836.252} C_VEL
LIN {X 0,Y 290.477,Z 908.84,A -85,B 0,C 180,E1 -16837.647,E2 -16837.647} C_VEL
LIN {X 0,Y 291.117,Z 903.738,A -85,B 0,C 180,E1 -16839.729,E2 -16839.729} C_VEL
LIN {X 0,Y 291.976,Z 898.243,A -85,B 0,C 180,E1 -16841.454,E2 -16841.454} C_VEL
LIN {X 0,Y 293.072,Z 891.333,A -85,B 0,C 180,E1 -16843.168,E2 -16843.168} C_VEL
LIN {X 0,Y 294.166,Z 883.399,A -85,B 0,C 180,E1 -16844.705,E2 -16844.705} C_VEL
LIN {X 0,Y 295.083,Z 875.833,A -85,B 0,C 180,E1 -16845.896,E2 -16845.896} C_VEL
LIN {X 0,Y 296.099,Z 867.895,A -85,B 0,C 180,E1 -16846.903,E2 -16846.903} C_VEL
LIN {X 0,Y 296.94,Z 859.692,A -85,B 0,C 180,E1 -16847.742,E2 -16847.742} C_VEL
LIN {X 0,Y 297.645,Z 851.37,A -85,B 0,C 180,E1 -16848.41,E2 -16848.41} C_VEL
LIN {X 0,Y 298.136,Z 842.364,A -85,B 0,C 180,E1 -16848.958,E2 -16848.958} C_VEL
LIN {X 0,Y 298.492,Z 832.513,A -85,B 0,C 180,E1 -16849.36,E2 -16849.36} C_VEL
LIN {X 0,Y 299.425,Z 785.568,A -85,B 0,C 180,E1 -16850.5,E2 -16850.5} C_VEL
LIN {X 0,Y 295.753,Z 767.087,A -85,B 0,C 180,E1 -16851.24,E2 -16851.24} C_VEL
LIN {X 0,Y 292.833,Z 758.376,A -85,B 0,C 180,E1 -16851.72,E2 -16851.72} C_VEL
LIN {X 0,Y 292.645,Z 757.479,A -85,B 0,C 180,E1 -16851.925,E2 -16851.925} C_VEL
LIN {X 0,Y 291.436,Z 751.086,A -85,B 0,C 180,E1 -16854.724,E2 -16854.724} C_VEL
LIN {X 0,Y 291.346,Z 751.006,A -85,B 0,C 180,E1 -16858.846,E2 -16858.846} C_VEL
LIN {X 0,Y 291.34,Z 750.989,A -85,B 0,C 180,E1 -16862.402,E2 -16862.402} C_VEL
LIN {X 0,Y 291.362,Z 751.007,A -85,B 0,C 180,E1 -16865.374,E2 -16865.374} C_VEL
LIN {X 0,Y 291.348,Z 750.976,A -85,B 0,C 180,E1 -16868.842,E2 -16868.842} C_VEL
LIN {X 0,Y 291.321,Z 751.012,A -85,B 0,C 180,E1 -16872.492,E2 -16872.492} C_VEL
LIN {X 0,Y 291.31,Z 750.963,A -85,B 0,C 180,E1 -16876.366,E2 -16876.366} C_VEL
LIN {X 0,Y 291.382,Z 750.982,A -85,B 0,C 180,E1 -16880.518,E2 -16880.518} C_VEL
LIN {X 0,Y 291.409,Z 751,A -85,B 0,C 180,E1 -16882.92,E2 -16882.92} C_VEL
LIN {X 0,Y 291.346,Z 750.99,A -85,B 0,C 180,E1 -16886.302,E2 -16886.302} C_VEL
LIN {X 0,Y 291.385,Z 751,A -85,B 0,C 180,E1 -16890.261,E2 -16890.261} C_VEL
LIN {X 0,Y 291.412,Z 750.974,A -85,B 0,C 180,E1 -16894.271,E2 -16894.271} C_VEL
LIN {X 0,Y 291.375,Z 751.001,A -85,B 0,C 180,E1 -16897.287,E2 -16897.287} C_VEL
LIN {X 0,Y 290.735,Z 751.089,A -85,B 0,C 180,E1 -16898.442,E2 -16898.442} C_VEL
LIN {X 0,Y 287.896,Z 751.43,A -85,B 0,C 180,E1 -16900.323,E2 -16900.323} C_VEL
LIN {X 0,Y 285.482,Z 751.715,A -85,B 0,C 180,E1 -16901.85,E2 -16901.85} C_VEL
LIN {X 0,Y 284.46,Z 751.837,A -85,B 0,C 180,E1 -16903.034,E2 -16903.034} C_VEL
LIN {X 0,Y 284.386,Z 751.848,A -85,B 0,C 180,E1 -16903.434,E2 -16903.434} C_VEL
LIN {X 0,Y 284.476,Z 751.862,A -85,B 0,C 180,E1 -16907.153,E2 -16907.153} C_VEL
LIN {X 0,Y 284.66,Z 751.81,A -85,B 0,C 180,E1 -16911.481,E2 -16911.481} C_VEL
LIN {X 0,Y 284.603,Z 751.831,A -85,B 0,C 180,E1 -16914.331,E2 -16914.331} C_VEL
LIN {X 0,Y 284.86,Z 751.81,A -85,B 0,C 180,E1 -16918.586,E2 -16918.586} C_VEL
LIN {X 0,Y 284.856,Z 751.786,A -85,B 0,C 180,E1 -16921.414,E2 -16921.414} C_VEL
LIN {X 0,Y 284.69,Z 751.834,A -85,B 0,C 180,E1 -16927.09,E2 -16927.09} C_VEL
LIN {X 0,Y 284.568,Z 751.837,A -85,B 0,C 180,E1 -16929.955,E2 -16929.955} C_VEL
LIN {X 0,Y 284.483,Z 751.848,A -85,B 0,C 180,E1 -16934.303,E2 -16934.303} C_VEL
LIN {X 0,Y 284.427,Z 751.867,A -85,B 0,C 180,E1 -16937.248,E2 -16937.248} C_VEL
LIN {X 0,Y 284.38,Z 751.852,A -85,B 0,C 180,E1 -16940.242,E2 -16940.242} C_VEL
LIN {X 0,Y 284.371,Z 751.868,A -85,B 0,C 180,E1 -16943.876,E2 -16943.876} C_VEL
LIN {X 0,Y 284.396,Z 751.867,A -85,B 0,C 180,E1 -16947.173,E2 -16947.173} C_VEL
LIN {X 0,Y 284.295,Z 751.877,A -85,B 0,C 180,E1 -16951.274,E2 -16951.274} C_VEL
LIN {X 0,Y 284.362,Z 751.866,A -85,B 0,C 180,E1 -16955.354,E2 -16955.354} C_VEL
LIN {X 0,Y 284.329,Z 751.823,A -85,B 0,C 180,E1 -16958.166,E2 -16958.166} C_VEL
LIN {X 0,Y 284.302,Z 751.855,A -85,B 0,C 180,E1 -16961.87,E2 -16961.87} C_VEL
LIN {X 0,Y 284.257,Z 751.883,A -85,B 0,C 180,E1 -16966.19,E2 -16966.19} C_VEL
LIN {X 0,Y 284.307,Z 751.868,A -85,B 0,C 180,E1 -16970.024,E2 -16970.024} C_VEL
LIN {X 0,Y 284.35,Z 751.865,A -85,B 0,C 180,E1 -16973.617,E2 -16973.617} C_VEL
LIN {X 0,Y 284.308,Z 751.872,A -85,B 0,C 180,E1 -16977.189,E2 -16977.189} C_VEL
LIN {X 0,Y 284.389,Z 752.055,A -85,B 0,C 180,E1 -16979.785,E2 -16979.785} C_VEL
LIN {X 0,Y 286.032,Z 760.228,A -85,B 0,C 180,E1 -16983.06,E2 -16983.06} C_VEL
LIN {X 0,Y 287.261,Z 767.421,A -85,B 0,C 180,E1 -16985.808,E2 -16985.808} C_VEL
LIN {X 0,Y 286.605,Z 773.144,A -85,B 0,C 180,E1 -16987.755,E2 -16987.755} C_VEL
LIN {X 0,Y 287.332,Z 777.425,A -85,B 0,C 180,E1 -16988.004,E2 -16988.004} C_VEL
LIN {X 0,Y 291.147,Z 801.605,A -85,B 0,C 180,E1 -16988.93,E2 -16988.93} C_VEL
LIN {X 0,Y 292.346,Z 812.31,A -85,B 0,C 180,E1 -16989.295,E2 -16989.295} C_VEL
LIN {X 0,Y 291.463,Z 850.883,A -85,B 0,C 180,E1 -16990.271,E2 -16990.271} C_VEL
LIN {X 0,Y 290.83,Z 861.682,A -85,B 0,C 180,E1 -16990.755,E2 -16990.755} C_VEL
LIN {X 0,Y 289.785,Z 873.764,A -85,B 0,C 180,E1 -16991.622,E2 -16991.622} C_VEL
LIN {X 0,Y 288.913,Z 882.461,A -85,B 0,C 180,E1 -16992.481,E2 -16992.481} C_VEL
LIN {X 0,Y 287.848,Z 890.768,A -85,B 0,C 180,E1 -16993.511,E2 -16993.511} C_VEL
LIN {X 0,Y 286.751,Z 898.633,A -85,B 0,C 180,E1 -16994.724,E2 -16994.724} C_VEL
LIN {X 0,Y 285.614,Z 905.989,A -85,B 0,C 180,E1 -16996.118,E2 -16996.118} C_VEL
LIN {X 0,Y 284.53,Z 913.457,A -85,B 0,C 180,E1 -16997.88,E2 -16997.88} C_VEL
LIN {X 0,Y 283.543,Z 920.276,A -85,B 0,C 180,E1 -17000.008,E2 -17000.008} C_VEL
LIN {X 0,Y 282.882,Z 925.46,A -85,B 0,C 180,E1 -17002.146,E2 -17002.146} C_VEL
LIN {X 0,Y 282.505,Z 929.324,A -85,B 0,C 180,E1 -17004.323,E2 -17004.323} C_VEL
LIN {X 0,Y 282.394,Z 931.02,A -85,B 0,C 180,E1 -17005.718,E2 -17005.718} C_VEL
LIN {X 0,Y 282.36,Z 932.275,A -85,B 0,C 180,E1 -17007.147,E2 -17007.147} C_VEL
LIN {X 0,Y 282.338,Z 933.055,A -85,B 0,C 180,E1 -17008.574,E2 -17008.574} C_VEL
LIN {X 0,Y 282.355,Z 933.35,A -85,B 0,C 180,E1 -17010,E2 -17010} C_VEL
LIN {X 0,Y 282.338,Z 933.05,A -85,B 0,C 180,E1 -17011.426,E2 -17011.426} C_VEL
LIN {X 0,Y 282.36,Z 932.26,A -85,B 0,C 180,E1 -17012.853,E2 -17012.853} C_VEL
LIN {X 0,Y 282.394,Z 930.994,A -85,B 0,C 180,E1 -17014.282,E2 -17014.282} C_VEL
LIN {X 0,Y 282.602,Z 928.072,A -85,B 0,C 180,E1 -17016.425,E2 -17016.425} C_VEL
LIN {X 0,Y 282.882,Z 925.412,A -85,B 0,C 180,E1 -17017.854,E2 -17017.854} C_VEL
LIN {X 0,Y 283.539,Z 920.212,A -85,B 0,C 180,E1 -17019.992,E2 -17019.992} C_VEL
LIN {X 0,Y 284.529,Z 913.363,A -85,B 0,C 180,E1 -17022.12,E2 -17022.12} C_VEL
LIN {X 0,Y 285.613,Z 905.881,A -85,B 0,C 180,E1 -17023.882,E2 -17023.882} C_VEL
LIN {X 0,Y 286.732,Z 898.507,A -85,B 0,C 180,E1 -17025.277,E2 -17025.277} C_VEL
LIN {X 0,Y 287.844,Z 890.611,A -85,B 0,C 180,E1 -17026.489,E2 -17026.489} C_VEL
LIN {X 0,Y 288.931,Z 882.266,A -85,B 0,C 180,E1 -17027.518,E2 -17027.518} C_VEL
LIN {X 0,Y 289.942,Z 871.603,A -85,B 0,C 180,E1 -17028.55,E2 -17028.55} C_VEL
LIN {X 0,Y 290.921,Z 860.031,A -85,B 0,C 180,E1 -17029.305,E2 -17029.305} C_VEL
LIN {X 0,Y 291.458,Z 850.198,A -85,B 0,C 180,E1 -17029.73,E2 -17029.73} C_VEL
LIN {X 0,Y 292.178,Z 809.601,A -85,B 0,C 180,E1 -17030.762,E2 -17030.762} C_VEL
LIN {X 0,Y 288.742,Z 785.577,A -85,B 0,C 180,E1 -17031.645,E2 -17031.645} C_VEL
LIN {X 0,Y 286.605,Z 773.546,A -85,B 0,C 180,E1 -17032.163,E2 -17032.163} C_VEL
LIN {X 0,Y 286.67,Z 772.462,A -85,B 0,C 180,E1 -17032.41,E2 -17032.41} C_VEL
LIN {X 0,Y 287.261,Z 767.354,A -85,B 0,C 180,E1 -17034.192,E2 -17034.192} C_VEL
LIN {X 0,Y 286.049,Z 760.177,A -85,B 0,C 180,E1 -17036.934,E2 -17036.934} C_VEL
LIN {X 0,Y 284.365,Z 751.912,A -85,B 0,C 180,E1 -17040.298,E2 -17040.298} C_VEL
LIN {X 0,Y 284.324,Z 751.876,A -85,B 0,C 180,E1 -17044.647,E2 -17044.647} C_VEL
LIN {X 0,Y 284.324,Z 751.881,A -85,B 0,C 180,E1 -17048.167,E2 -17048.167} C_VEL
LIN {X 0,Y 284.269,Z 751.865,A -85,B 0,C 180,E1 -17052.124,E2 -17052.124} C_VEL
LIN {X 0,Y 284.274,Z 751.882,A -85,B 0,C 180,E1 -17056.193,E2 -17056.193} C_VEL
LIN {X 0,Y 284.352,Z 751.814,A -85,B 0,C 180,E1 -17060.013,E2 -17060.013} C_VEL
LIN {X 0,Y 284.353,Z 751.853,A -85,B 0,C 180,E1 -17063.617,E2 -17063.617} C_VEL
LIN {X 0,Y 284.308,Z 751.882,A -85,B 0,C 180,E1 -17067.19,E2 -17067.19} C_VEL
LIN {X 0,Y 284.356,Z 751.856,A -85,B 0,C 180,E1 -17070.376,E2 -17070.376} C_VEL
LIN {X 0,Y 284.377,Z 751.872,A -85,B 0,C 180,E1 -17073.587,E2 -17073.587} C_VEL
LIN {X 0,Y 284.368,Z 751.863,A -85,B 0,C 180,E1 -17076.707,E2 -17076.707} C_VEL
LIN {X 0,Y 284.406,Z 751.864,A -85,B 0,C 180,E1 -17081.262,E2 -17081.262} C_VEL
LIN {X 0,Y 284.493,Z 751.854,A -85,B 0,C 180,E1 -17084.459,E2 -17084.459} C_VEL
LIN {X 0,Y 284.489,Z 751.834,A -85,B 0,C 180,E1 -17088.602,E2 -17088.602} C_VEL
LIN {X 0,Y 284.651,Z 751.836,A -85,B 0,C 180,E1 -17091.481,E2 -17091.481} C_VEL
LIN {X 0,Y 284.599,Z 751.841,A -85,B 0,C 180,E1 -17094.331,E2 -17094.331} C_VEL
LIN {X 0,Y 284.857,Z 751.785,A -85,B 0,C 180,E1 -17098.586,E2 -17098.586} C_VEL
LIN {X 0,Y 284.86,Z 751.81,A -85,B 0,C 180,E1 -17101.414,E2 -17101.414} C_VEL
LIN {X 0,Y 284.7,Z 751.802,A -85,B 0,C 180,E1 -17107.09,E2 -17107.09} C_VEL
LIN {X 0,Y 284.568,Z 751.838,A -85,B 0,C 180,E1 -17109.955,E2 -17109.955} C_VEL
LIN {X 0,Y 284.469,Z 751.859,A -85,B 0,C 180,E1 -17114.304,E2 -17114.304} C_VEL
LIN {X 0,Y 284.384,Z 751.854,A -85,B 0,C 180,E1 -17118.74,E2 -17118.74} C_VEL
LIN {X 0,Y 284.318,Z 751.88,A -85,B 0,C 180,E1 -17121.764,E2 -17121.764} C_VEL
LIN {X 0,Y 284.338,Z 751.86,A -85,B 0,C 180,E1 -17124.847,E2 -17124.847} C_VEL
LIN {X 0,Y 284.329,Z 751.874,A -85,B 0,C 180,E1 -17128.011,E2 -17128.011} C_VEL
LIN {X 0,Y 284.295,Z 751.879,A -85,B 0,C 180,E1 -17131.275,E2 -17131.275} C_VEL
LIN {X 0,Y 284.342,Z 751.873,A -85,B 0,C 180,E1 -17135.348,E2 -17135.348} C_VEL
LIN {X 0,Y 284.313,Z 751.878,A -85,B 0,C 180,E1 -17138.169,E2 -17138.169} C_VEL
LIN {X 0,Y 284.269,Z 751.83,A -85,B 0,C 180,E1 -17142.124,E2 -17142.124} C_VEL
LIN {X 0,Y 284.257,Z 751.883,A -85,B 0,C 180,E1 -17146.189,E2 -17146.189} C_VEL
LIN {X 0,Y 284.307,Z 751.866,A -85,B 0,C 180,E1 -17150.024,E2 -17150.024} C_VEL
LIN {X 0,Y 284.332,Z 751.869,A -85,B 0,C 180,E1 -17153.614,E2 -17153.614} C_VEL
LIN {X 0,Y 284.307,Z 751.87,A -85,B 0,C 180,E1 -17157.19,E2 -17157.19} C_VEL
LIN {X 0,Y 284.338,Z 751.88,A -85,B 0,C 180,E1 -17160.374,E2 -17160.374} C_VEL
LIN {X 0,Y 284.38,Z 751.941,A -85,B 0,C 180,E1 -17164.962,E2 -17164.962} C_VEL
LIN {X 0,Y 284.405,Z 752.109,A -85,B 0,C 180,E1 -17165.16,E2 -17165.16} C_VEL
LIN {X 0,Y 285.527,Z 758.007,A -85,B 0,C 180,E1 -17167.719,E2 -17167.719} C_VEL
LIN {X 0,Y 285.991,Z 759.662,A -85,B 0,C 180,E1 -17167.907,E2 -17167.907} C_VEL
LIN {X 0,Y 289.599,Z 770.174,A -85,B 0,C 180,E1 -17168.478,E2 -17168.478} C_VEL
LIN {X 0,Y 292.753,Z 787.07,A -85,B 0,C 180,E1 -17169.16,E2 -17169.16} C_VEL
LIN {X 0,Y 291.741,Z 834.064,A -85,B 0,C 180,E1 -17170.336,E2 -17170.336} C_VEL
LIN {X 0,Y 291.39,Z 843.807,A -85,B 0,C 180,E1 -17170.769,E2 -17170.769} C_VEL
LIN {X 0,Y 290.518,Z 854.871,A -85,B 0,C 180,E1 -17171.488,E2 -17171.488} C_VEL
LIN {X 0,Y 289.592,Z 865.662,A -85,B 0,C 180,E1 -17172.523,E2 -17172.523} C_VEL
LIN {X 0,Y 288.48,Z 874.045,A -85,B 0,C 180,E1 -17173.548,E2 -17173.548} C_VEL
LIN {X 0,Y 287.519,Z 881.953,A -85,B 0,C 180,E1 -17174.766,E2 -17174.766} C_VEL
LIN {X 0,Y 286.422,Z 889.329,A -85,B 0,C 180,E1 -17176.158,E2 -17176.158} C_VEL
LIN {X 0,Y 285.296,Z 896.797,A -85,B 0,C 180,E1 -17177.913,E2 -17177.913} C_VEL
LIN {X 0,Y 284.192,Z 903.641,A -85,B 0,C 180,E1 -17180.031,E2 -17180.031} C_VEL
LIN {X 0,Y 283.455,Z 908.809,A -85,B 0,C 180,E1 -17182.162,E2 -17182.162} C_VEL
LIN {X 0,Y 283.184,Z 910.649,A -85,B 0,C 180,E1 -17183.08,E2 -17183.08} C_VEL
LIN {X 0,Y 282.967,Z 912.603,A -85,B 0,C 180,E1 -17184.298,E2 -17184.298} C_VEL
LIN {X 0,Y 282.702,Z 914.362,A -85,B 0,C 180,E1 -17185.723,E2 -17185.723} C_VEL
LIN {X 0,Y 282.516,Z 915.629,A -85,B 0,C 180,E1 -17187.148,E2 -17187.148} C_VEL
LIN {X 0,Y 282.386,Z 916.429,A -85,B 0,C 180,E1 -17188.574,E2 -17188.574} C_VEL
LIN {X 0,Y 282.363,Z 916.733,A -85,B 0,C 180,E1 -17190,E2 -17190} C_VEL
LIN {X 0,Y 282.383,Z 916.454,A -85,B 0,C 180,E1 -17191.426,E2 -17191.426} C_VEL
LIN {X 0,Y 282.509,Z 915.706,A -85,B 0,C 180,E1 -17192.852,E2 -17192.852} C_VEL
LIN {X 0,Y 282.699,Z 914.491,A -85,B 0,C 180,E1 -17194.277,E2 -17194.277} C_VEL
LIN {X 0,Y 282.94,Z 912.786,A -85,B 0,C 180,E1 -17195.702,E2 -17195.702} C_VEL
LIN {X 0,Y 283.442,Z 909.048,A -85,B 0,C 180,E1 -17197.838,E2 -17197.838} C_VEL
LIN {X 0,Y 284.125,Z 903.945,A -85,B 0,C 180,E1 -17199.971,E2 -17199.971} C_VEL
LIN {X 0,Y 285.028,Z 898.449,A -85,B 0,C 180,E1 -17201.737,E2 -17201.737} C_VEL
LIN {X 0,Y 286.182,Z 891.539,A -85,B 0,C 180,E1 -17203.491,E2 -17203.491} C_VEL
LIN {X 0,Y 287.315,Z 883.604,A -85,B 0,C 180,E1 -17205.064,E2 -17205.064} C_VEL
LIN {X 0,Y 288.285,Z 876.037,A -85,B 0,C 180,E1 -17206.281,E2 -17206.281} C_VEL
LIN {X 0,Y 289.31,Z 868.098,A -85,B 0,C 180,E1 -17207.312,E2 -17207.312} C_VEL
LIN {X 0,Y 290.202,Z 859.894,A -85,B 0,C 180,E1 -17208.168,E2 -17208.168} C_VEL
LIN {X 0,Y 290.942,Z 851.57,A -85,B 0,C 180,E1 -17208.85,E2 -17208.85} C_VEL
LIN {X 0,Y 291.444,Z 842.561,A -85,B 0,C 180,E1 -17209.41,E2 -17209.41} C_VEL
LIN {X 0,Y 291.793,Z 833.401,A -85,B 0,C 180,E1 -17209.798,E2 -17209.798} C_VEL
LIN {X 0,Y 292.729,Z 786.244,A -85,B 0,C 180,E1 -17210.978,E2 -17210.978} C_VEL
LIN {X 0,Y 289.352,Z 769.16,A -85,B 0,C 180,E1 -17211.684,E2 -17211.684} C_VEL
LIN {X 0,Y 285.677,Z 758.509,A -85,B 0,C 180,E1 -17212.303,E2 -17212.303} C_VEL
LIN {X 0,Y 285.435,Z 757.35,A -85,B 0,C 180,E1 -17212.634,E2 -17212.634} C_VEL
LIN {X 0,Y 284.406,Z 751.965,A -85,B 0,C 180,E1 -17215.084,E2 -17215.084} C_VEL
LIN {X 0,Y 284.338,Z 751.88,A -85,B 0,C 180,E1 -17219.626,E2 -17219.626} C_VEL
LIN {X 0,Y 284.305,Z 751.87,A -85,B 0,C 180,E1 -17222.945,E2 -17222.945} C_VEL
LIN {X 0,Y 284.332,Z 751.871,A -85,B 0,C 180,E1 -17226.386,E2 -17226.386} C_VEL
LIN {X 0,Y 284.307,Z 751.863,A -85,B 0,C 180,E1 -17229.995,E2 -17229.995} C_VEL
LIN {X 0,Y 284.247,Z 751.88,A -85,B 0,C 180,E1 -17234.19,E2 -17234.19} C_VEL
LIN {X 0,Y 284.272,Z 751.831,A -85,B 0,C 180,E1 -17238.124,E2 -17238.124} C_VEL
LIN {X 0,Y 284.324,Z 751.877,A -85,B 0,C 180,E1 -17242.278,E2 -17242.278} C_VEL
LIN {X 0,Y 284.31,Z 751.872,A -85,B 0,C 180,E1 -17245.351,E2 -17245.351} C_VEL
LIN {X 0,Y 284.295,Z 751.878,A -85,B 0,C 180,E1 -17248.725,E2 -17248.725} C_VEL
LIN {X 0,Y 284.396,Z 751.856,A -85,B 0,C 180,E1 -17252.827,E2 -17252.827} C_VEL
LIN {X 0,Y 284.334,Z 751.872,A -85,B 0,C 180,E1 -17256.704,E2 -17256.704} C_VEL
LIN {X 0,Y 284.389,Z 751.867,A -85,B 0,C 180,E1 -17259.898,E2 -17259.898} C_VEL
LIN {X 0,Y 284.386,Z 751.848,A -85,B 0,C 180,E1 -17263.434,E2 -17263.434} C_VEL
LIN {X 0,Y 283.734,Z 751.939,A -85,B 0,C 180,E1 -17264.616,E2 -17264.616} C_VEL
LIN {X 0,Y 280.882,Z 752.306,A -85,B 0,C 180,E1 -17266.542,E2 -17266.542} C_VEL
LIN {X 0,Y 278.5,Z 752.604,A -85,B 0,C 180,E1 -17268.107,E2 -17268.107} C_VEL
LIN {X 0,Y 277.544,Z 752.718,A -85,B 0,C 180,E1 -17269.319,E2 -17269.319} C_VEL
LIN {X 0,Y 277.502,Z 752.72,A -85,B 0,C 180,E1 -17269.729,E2 -17269.729} C_VEL
LIN {X 0,Y 277.655,Z 752.678,A -85,B 0,C 180,E1 -17272.729,E2 -17272.729} C_VEL
LIN {X 0,Y 277.826,Z 752.686,A -85,B 0,C 180,E1 -17278.55,E2 -17278.55} C_VEL
LIN {X 0,Y 277.822,Z 752.661,A -85,B 0,C 180,E1 -17281.449,E2 -17281.449} C_VEL
LIN {X 0,Y 277.645,Z 752.712,A -85,B 0,C 180,E1 -17287.271,E2 -17287.271} C_VEL
LIN {X 0,Y 277.508,Z 752.714,A -85,B 0,C 180,E1 -17290.211,E2 -17290.211} C_VEL
LIN {X 0,Y 277.436,Z 752.731,A -85,B 0,C 180,E1 -17294.674,E2 -17294.674} C_VEL
LIN {X 0,Y 277.348,Z 752.74,A -85,B 0,C 180,E1 -17299.233,E2 -17299.233} C_VEL
LIN {X 0,Y 277.321,Z 752.749,A -85,B 0,C 180,E1 -17304.17,E2 -17304.17} C_VEL
LIN {X 0,Y 277.324,Z 752.746,A -85,B 0,C 180,E1 -17307.504,E2 -17307.504} C_VEL
LIN {X 0,Y 277.272,Z 752.743,A -85,B 0,C 180,E1 -17310.481,E2 -17310.481} C_VEL
LIN {X 0,Y 277.255,Z 752.762,A -85,B 0,C 180,E1 -17313.894,E2 -17313.894} C_VEL
LIN {X 0,Y 277.285,Z 752.71,A -85,B 0,C 180,E1 -17317.466,E2 -17317.466} C_VEL
LIN {X 0,Y 277.24,Z 752.717,A -85,B 0,C 180,E1 -17321.231,E2 -17321.231} C_VEL
LIN {X 0,Y 277.206,Z 752.766,A -85,B 0,C 180,E1 -17325.225,E2 -17325.225} C_VEL
LIN {X 0,Y 277.222,Z 752.743,A -85,B 0,C 180,E1 -17329.512,E2 -17329.512} C_VEL
LIN {X 0,Y 277.282,Z 752.754,A -85,B 0,C 180,E1 -17332.533,E2 -17332.533} C_VEL
LIN {X 0,Y 277.254,Z 752.763,A -85,B 0,C 180,E1 -17336.105,E2 -17336.105} C_VEL
LIN {X 0,Y 277.339,Z 752.934,A -85,B 0,C 180,E1 -17339.359,E2 -17339.359} C_VEL
LIN {X 0,Y 279.138,Z 761.873,A -85,B 0,C 180,E1 -17343.051,E2 -17343.051} C_VEL
LIN {X 0,Y 280.237,Z 768.27,A -85,B 0,C 180,E1 -17345.556,E2 -17345.556} C_VEL
LIN {X 0,Y 279.824,Z 772.737,A -85,B 0,C 180,E1 -17347.137,E2 -17347.137} C_VEL
LIN {X 0,Y 280.019,Z 774.757,A -85,B 0,C 180,E1 -17347.328,E2 -17347.328} C_VEL
LIN {X 0,Y 283.779,Z 796.772,A -85,B 0,C 180,E1 -17348.233,E2 -17348.233} C_VEL
LIN {X 0,Y 285.711,Z 812.4,A -85,B 0,C 180,E1 -17348.799,E2 -17348.799} C_VEL
LIN {X 0,Y 284.786,Z 850.69,A -85,B 0,C 180,E1 -17349.788,E2 -17349.788} C_VEL
LIN {X 0,Y 284.154,Z 861.302,A -85,B 0,C 180,E1 -17350.275,E2 -17350.275} C_VEL
LIN {X 0,Y 283.065,Z 873.561,A -85,B 0,C 180,E1 -17351.17,E2 -17351.17} C_VEL
LIN {X 0,Y 282.145,Z 882.256,A -85,B 0,C 180,E1 -17352.046,E2 -17352.046} C_VEL
LIN {X 0,Y 281.054,Z 890.563,A -85,B 0,C 180,E1 -17353.101,E2 -17353.101} C_VEL
LIN {X 0,Y 279.914,Z 898.428,A -85,B 0,C 180,E1 -17354.341,E2 -17354.341} C_VEL
LIN {X 0,Y 278.726,Z 905.783,A -85,B 0,C 180,E1 -17355.768,E2 -17355.768} C_VEL
LIN {X 0,Y 277.589,Z 913.25,A -85,B 0,C 180,E1 -17357.573,E2 -17357.573} C_VEL
LIN {X 0,Y 276.541,Z 920.068,A -85,B 0,C 180,E1 -17359.753,E2 -17359.753} C_VEL
LIN {X 0,Y 275.823,Z 925.251,A -85,B 0,C 180,E1 -17361.944,E2 -17361.944} C_VEL
LIN {X 0,Y 275.525,Z 927.901,A -85,B 0,C 180,E1 -17363.409,E2 -17363.409} C_VEL
LIN {X 0,Y 275.425,Z 929.386,A -85,B 0,C 180,E1 -17364.359,E2 -17364.359} C_VEL
LIN {X 0,Y 275.272,Z 932.067,A -85,B 0,C 180,E1 -17367.073,E2 -17367.073} C_VEL
LIN {X 0,Y 275.263,Z 932.847,A -85,B 0,C 180,E1 -17368.537,E2 -17368.537} C_VEL
LIN {X 0,Y 275.277,Z 933.142,A -85,B 0,C 180,E1 -17370,E2 -17370} C_VEL
LIN {X 0,Y 275.263,Z 932.841,A -85,B 0,C 180,E1 -17371.463,E2 -17371.463} C_VEL
LIN {X 0,Y 275.272,Z 932.05,A -85,B 0,C 180,E1 -17372.927,E2 -17372.927} C_VEL
LIN {X 0,Y 275.405,Z 929.411,A -85,B 0,C 180,E1 -17375.598,E2 -17375.598} C_VEL
LIN {X 0,Y 275.691,Z 926.687,A -85,B 0,C 180,E1 -17377.323,E2 -17377.323} C_VEL
LIN {X 0,Y 276.261,Z 921.924,A -85,B 0,C 180,E1 -17379.518,E2 -17379.518} C_VEL
LIN {X 0,Y 277,Z 916.769,A -85,B 0,C 180,E1 -17381.34,E2 -17381.34} C_VEL
LIN {X 0,Y 277.819,Z 911.734,A -85,B 0,C 180,E1 -17382.788,E2 -17382.788} C_VEL
LIN {X 0,Y 278.725,Z 905.67,A -85,B 0,C 180,E1 -17384.232,E2 -17384.232} C_VEL
LIN {X 0,Y 279.889,Z 898.295,A -85,B 0,C 180,E1 -17385.66,E2 -17385.66} C_VEL
LIN {X 0,Y 281.053,Z 890.398,A -85,B 0,C 180,E1 -17386.9,E2 -17386.9} C_VEL
LIN {X 0,Y 282.16,Z 882.053,A -85,B 0,C 180,E1 -17387.953,E2 -17387.953} C_VEL
LIN {X 0,Y 283.226,Z 871.492,A -85,B 0,C 180,E1 -17388.997,E2 -17388.997} C_VEL
LIN {X 0,Y 284.234,Z 859.937,A -85,B 0,C 180,E1 -17389.771,E2 -17389.771} C_VEL
LIN {X 0,Y 284.75,Z 851.11,A -85,B 0,C 180,E1 -17390.173,E2 -17390.173} C_VEL
LIN {X 0,Y 285.359,Z 822.292,A -85,B 0,C 180,E1 -17390.941,E2 -17390.941} C_VEL
LIN {X 0,Y 285.53,Z 810.247,A -85,B 0,C 180,E1 -17391.246,E2 -17391.246} C_VEL
LIN {X 0,Y 282.16,Z 786.676,A -85,B 0,C 180,E1 -17392.141,E2 -17392.141} C_VEL
LIN {X 0,Y 279.805,Z 773.145,A -85,B 0,C 180,E1 -17392.754,E2 -17392.754} C_VEL
LIN {X 0,Y 280.303,Z 769.259,A -85,B 0,C 180,E1 -17394.044,E2 -17394.044} C_VEL
LIN {X 0,Y 279.358,Z 762.876,A -85,B 0,C 180,E1 -17396.522,E2 -17396.522} C_VEL
LIN {X 0,Y 277.382,Z 753.08,A -85,B 0,C 180,E1 -17400.52,E2 -17400.52} C_VEL
LIN {X 0,Y 277.313,Z 752.73,A -85,B 0,C 180,E1 -17400.876,E2 -17400.876} C_VEL
LIN {X 0,Y 277.325,Z 752.739,A -85,B 0,C 180,E1 -17405.812,E2 -17405.812} C_VEL
LIN {X 0,Y 277.238,Z 752.755,A -85,B 0,C 180,E1 -17409.327,E2 -17409.327} C_VEL
LIN {X 0,Y 277.21,Z 752.755,A -85,B 0,C 180,E1 -17413.198,E2 -17413.198} C_VEL
LIN {X 0,Y 277.237,Z 752.745,A -85,B 0,C 180,E1 -17417.32,E2 -17417.32} C_VEL
LIN {X 0,Y 277.266,Z 752.694,A -85,B 0,C 180,E1 -17420.677,E2 -17420.677} C_VEL
LIN {X 0,Y 277.305,Z 752.74,A -85,B 0,C 180,E1 -17424.345,E2 -17424.345} C_VEL
LIN {X 0,Y 277.244,Z 752.76,A -85,B 0,C 180,E1 -17427.837,E2 -17427.837} C_VEL
LIN {X 0,Y 277.269,Z 752.741,A -85,B 0,C 180,E1 -17431.21,E2 -17431.21} C_VEL
LIN {X 0,Y 277.314,Z 752.753,A -85,B 0,C 180,E1 -17434.48,E2 -17434.48} C_VEL
LIN {X 0,Y 277.288,Z 752.736,A -85,B 0,C 180,E1 -17437.655,E2 -17437.655} C_VEL
LIN {X 0,Y 277.347,Z 752.741,A -85,B 0,C 180,E1 -17440.767,E2 -17440.767} C_VEL
LIN {X 0,Y 277.436,Z 752.73,A -85,B 0,C 180,E1 -17445.326,E2 -17445.326} C_VEL
LIN {X 0,Y 277.508,Z 752.715,A -85,B 0,C 180,E1 -17449.789,E2 -17449.789} C_VEL
LIN {X 0,Y 277.645,Z 752.712,A -85,B 0,C 180,E1 -17452.729,E2 -17452.729} C_VEL
LIN {X 0,Y 277.823,Z 752.661,A -85,B 0,C 180,E1 -17458.551,E2 -17458.551} C_VEL
LIN {X 0,Y 277.826,Z 752.686,A -85,B 0,C 180,E1 -17461.45,E2 -17461.45} C_VEL
LIN {X 0,Y 277.655,Z 752.678,A -85,B 0,C 180,E1 -17467.271,E2 -17467.271} C_VEL
LIN {X 0,Y 277.508,Z 752.719,A -85,B 0,C 180,E1 -17470.211,E2 -17470.211} C_VEL
LIN {X 0,Y 277.416,Z 752.732,A -85,B 0,C 180,E1 -17474.675,E2 -17474.675} C_VEL
LIN {X 0,Y 277.33,Z 752.738,A -85,B 0,C 180,E1 -17479.235,E2 -17479.235} C_VEL
LIN {X 0,Y 277.298,Z 752.747,A -85,B 0,C 180,E1 -17483.923,E2 -17483.923} C_VEL
LIN {X 0,Y 277.324,Z 752.739,A -85,B 0,C 180,E1 -17487.504,E2 -17487.504} C_VEL
LIN {X 0,Y 277.273,Z 752.758,A -85,B 0,C 180,E1 -17490.481,E2 -17490.481} C_VEL
LIN {X 0,Y 277.248,Z 752.745,A -85,B 0,C 180,E1 -17493.896,E2 -17493.896} C_VEL
LIN {X 0,Y 277.269,Z 752.759,A -85,B 0,C 180,E1 -17497.469,E2 -17497.469} C_VEL
LIN {X 0,Y 277.21,Z 752.716,A -85,B 0,C 180,E1 -17501.237,E2 -17501.237} C_VEL
LIN {X 0,Y 277.202,Z 752.748,A -85,B 0,C 180,E1 -17505.227,E2 -17505.227} C_VEL
LIN {X 0,Y 277.224,Z 752.752,A -85,B 0,C 180,E1 -17509.512,E2 -17509.512} C_VEL
LIN {X 0,Y 277.265,Z 752.733,A -85,B 0,C 180,E1 -17512.53,E2 -17512.53} C_VEL
LIN {X 0,Y 277.248,Z 752.762,A -85,B 0,C 180,E1 -17516.104,E2 -17516.104} C_VEL
LIN {X 0,Y 277.263,Z 752.749,A -85,B 0,C 180,E1 -17519.539,E2 -17519.539} C_VEL
LIN {X 0,Y 277.294,Z 752.756,A -85,B 0,C 180,E1 -17522.857,E2 -17522.857} C_VEL
LIN {X 0,Y 277.344,Z 752.924,A -85,B 0,C 180,E1 -17524.735,E2 -17524.735} C_VEL
LIN {X 0,Y 278.333,Z 758.16,A -85,B 0,C 180,E1 -17527.094,E2 -17527.094} C_VEL
LIN {X 0,Y 278.729,Z 759.676,A -85,B 0,C 180,E1 -17527.29,E2 -17527.29} C_VEL
LIN {X 0,Y 282.903,Z 771.086,A -85,B 0,C 180,E1 -17527.96,E2 -17527.96} C_VEL
LIN {X 0,Y 286.049,Z 787.162,A -85,B 0,C 180,E1 -17528.644,E2 -17528.644} C_VEL
LIN {X 0,Y 285.075,Z 834.291,A -85,B 0,C 180,E1 -17529.856,E2 -17529.856} C_VEL
LIN {X 0,Y 284.716,Z 844.027,A -85,B 0,C 180,E1 -17530.3,E2 -17530.3} C_VEL
LIN {X 0,Y 283.811,Z 855.087,A -85,B 0,C 180,E1 -17531.034,E2 -17531.034} C_VEL
LIN {X 0,Y 282.841,Z 865.875,A -85,B 0,C 180,E1 -17532.092,E2 -17532.092} C_VEL
LIN {X 0,Y 281.692,Z 874.258,A -85,B 0,C 180,E1 -17533.14,E2 -17533.14} C_VEL
LIN {X 0,Y 280.688,Z 882.165,A -85,B 0,C 180,E1 -17534.385,E2 -17534.385} C_VEL
LIN {X 0,Y 279.862,Z 887.843,A -85,B 0,C 180,E1 -17535.456,E2 -17535.456} C_VEL
LIN {X 0,Y 278.806,Z 894.185,A -85,B 0,C 180,E1 -17536.887,E2 -17536.887} C_VEL
LIN {X 0,Y 277.932,Z 899.454,A -85,B 0,C 180,E1 -17538.329,E2 -17538.329} C_VEL
LIN {X 0,Y 277.198,Z 903.852,A -85,B 0,C 180,E1 -17539.777,E2 -17539.777} C_VEL
LIN {X 0,Y 276.433,Z 909.019,A -85,B 0,C 180,E1 -17541.962,E2 -17541.962} C_VEL
LIN {X 0,Y 276.108,Z 911.127,A -85,B 0,C 180,E1 -17543.074,E2 -17543.074} C_VEL
LIN {X 0,Y 275.895,Z 912.813,A -85,B 0,C 180,E1 -17544.152,E2 -17544.152} C_VEL
LIN {X 0,Y 275.631,Z 914.572,A -85,B 0,C 180,E1 -17545.613,E2 -17545.613} C_VEL
LIN {X 0,Y 275.451,Z 915.838,A -85,B 0,C 180,E1 -17547.075,E2 -17547.075} C_VEL
LIN {X 0,Y 275.312,Z 916.637,A -85,B 0,C 180,E1 -17548.537,E2 -17548.537} C_VEL
LIN {X 0,Y 275.285,Z 916.941,A -85,B 0,C 180,E1 -17550,E2 -17550} C_VEL
LIN {X 0,Y 275.309,Z 916.662,A -85,B 0,C 180,E1 -17551.463,E2 -17551.463} C_VEL
LIN {X 0,Y 275.445,Z 915.914,A -85,B 0,C 180,E1 -17552.925,E2 -17552.925} C_VEL
LIN {X 0,Y 275.627,Z 914.699,A -85,B 0,C 180,E1 -17554.387,E2 -17554.387} C_VEL
LIN {X 0,Y 275.871,Z 912.994,A -85,B 0,C 180,E1 -17555.849,E2 -17555.849} C_VEL
LIN {X 0,Y 276.4,Z 909.256,A -85,B 0,C 180,E1 -17558.039,E2 -17558.039} C_VEL
LIN {X 0,Y 277.129,Z 904.153,A -85,B 0,C 180,E1 -17560.225,E2 -17560.225} C_VEL
LIN {X 0,Y 278.096,Z 898.656,A -85,B 0,C 180,E1 -17562.034,E2 -17562.034} C_VEL
LIN {X 0,Y 279.302,Z 891.745,A -85,B 0,C 180,E1 -17563.83,E2 -17563.83} C_VEL
LIN {X 0,Y 280.47,Z 883.81,A -85,B 0,C 180,E1 -17565.441,E2 -17565.441} C_VEL
LIN {X 0,Y 281.48,Z 876.242,A -85,B 0,C 180,E1 -17566.686,E2 -17566.686} C_VEL
LIN {X 0,Y 282.558,Z 868.302,A -85,B 0,C 180,E1 -17567.74,E2 -17567.74} C_VEL
LIN {X 0,Y 283.469,Z 860.096,A -85,B 0,C 180,E1 -17568.615,E2 -17568.615} C_VEL
LIN {X 0,Y 284.257,Z 851.77,A -85,B 0,C 180,E1 -17569.31,E2 -17569.31} C_VEL
LIN {X 0,Y 284.781,Z 842.758,A -85,B 0,C 180,E1 -17569.883,E2 -17569.883} C_VEL
LIN {X 0,Y 285.15,Z 833.519,A -85,B 0,C 180,E1 -17570.282,E2 -17570.282} C_VEL
LIN {X 0,Y 286.058,Z 786.763,A -85,B 0,C 180,E1 -17571.482,E2 -17571.482} C_VEL
LIN {X 0,Y 282.964,Z 771.231,A -85,B 0,C 180,E1 -17572.148,E2 -17572.148} C_VEL
LIN {X 0,Y 278.531,Z 758.753,A -85,B 0,C 180,E1 -17572.903,E2 -17572.903} C_VEL
LIN {X 0,Y 278.317,Z 757.753,A -85,B 0,C 180,E1 -17573.175,E2 -17573.175} C_VEL
LIN {X 0,Y 277.339,Z 752.829,A -85,B 0,C 180,E1 -17575.518,E2 -17575.518} C_VEL
LIN {X 0,Y 277.241,Z 752.762,A -85,B 0,C 180,E1 -17578.793,E2 -17578.793} C_VEL
LIN {X 0,Y 277.241,Z 752.744,A -85,B 0,C 180,E1 -17582.164,E2 -17582.164} C_VEL
LIN {X 0,Y 277.281,Z 752.758,A -85,B 0,C 180,E1 -17585.799,E2 -17585.799} C_VEL
LIN {X 0,Y 277.234,Z 752.735,A -85,B 0,C 180,E1 -17589.328,E2 -17589.328} C_VEL
LIN {X 0,Y 277.211,Z 752.765,A -85,B 0,C 180,E1 -17593.198,E2 -17593.198} C_VEL
LIN {X 0,Y 277.215,Z 752.708,A -85,B 0,C 180,E1 -17597.325,E2 -17597.325} C_VEL
LIN {X 0,Y 277.266,Z 752.755,A -85,B 0,C 180,E1 -17601.792,E2 -17601.792} C_VEL
LIN {X 0,Y 277.286,Z 752.757,A -85,B 0,C 180,E1 -17604.341,E2 -17604.341} C_VEL
LIN {X 0,Y 277.245,Z 752.751,A -85,B 0,C 180,E1 -17607.836,E2 -17607.836} C_VEL
LIN {X 0,Y 277.269,Z 752.757,A -85,B 0,C 180,E1 -17611.21,E2 -17611.21} C_VEL
LIN {X 0,Y 277.308,Z 752.73,A -85,B 0,C 180,E1 -17614.479,E2 -17614.479} C_VEL
LIN {X 0,Y 277.269,Z 752.759,A -85,B 0,C 180,E1 -17617.653,E2 -17617.653} C_VEL
LIN {X 0,Y 277.336,Z 752.739,A -85,B 0,C 180,E1 -17620.765,E2 -17620.765} C_VEL
LIN {X 0,Y 277.416,Z 752.731,A -85,B 0,C 180,E1 -17625.325,E2 -17625.325} C_VEL
LIN {X 0,Y 277.502,Z 752.72,A -85,B 0,C 180,E1 -17629.729,E2 -17629.729} C_VEL
LIN {X 0,Y 276.901,Z 752.796,A -85,B 0,C 180,E1 -17630.942,E2 -17630.942} C_VEL
LIN {X 0,Y 273.984,Z 753.159,A -85,B 0,C 180,E1 -17632.916,E2 -17632.916} C_VEL
LIN {X 0,Y 271.512,Z 753.466,A -85,B 0,C 180,E1 -17634.521,E2 -17634.521} C_VEL
LIN {X 0,Y 270.531,Z 753.594,A -85,B 0,C 180,E1 -17635.768,E2 -17635.768} C_VEL
LIN {X 0,Y 270.497,Z 753.595,A -85,B 0,C 180,E1 -17636.19,E2 -17636.19} C_VEL
LIN {X 0,Y 270.792,Z 753.562,A -85,B 0,C 180,E1 -17638.513,E2 -17638.513} C_VEL
LIN {X 0,Y 270.788,Z 753.536,A -85,B 0,C 180,E1 -17641.487,E2 -17641.487} C_VEL
LIN {X 0,Y 270.604,Z 753.591,A -85,B 0,C 180,E1 -17647.461,E2 -17647.461} C_VEL
LIN {X 0,Y 270.443,Z 753.593,A -85,B 0,C 180,E1 -17650.481,E2 -17650.481} C_VEL
LIN {X 0,Y 270.404,Z 753.607,A -85,B 0,C 180,E1 -17655.064,E2 -17655.064} C_VEL
LIN {X 0,Y 270.304,Z 753.609,A -85,B 0,C 180,E1 -17659.755,E2 -17659.755} C_VEL
LIN {X 0,Y 270.275,Z 753.63,A -85,B 0,C 180,E1 -17664.585,E2 -17664.585} C_VEL
LIN {X 0,Y 270.27,Z 753.618,A -85,B 0,C 180,E1 -17667.909,E2 -17667.909} C_VEL
LIN {X 0,Y 270.185,Z 753.635,A -85,B 0,C 180,E1 -17671.348,E2 -17671.348} C_VEL
LIN {X 0,Y 270.216,Z 753.63,A -85,B 0,C 180,E1 -17674.903,E2 -17674.903} C_VEL
LIN {X 0,Y 270.223,Z 753.572,A -85,B 0,C 180,E1 -17678.717,E2 -17678.717} C_VEL
LIN {X 0,Y 270.192,Z 753.621,A -85,B 0,C 180,E1 -17682.554,E2 -17682.554} C_VEL
LIN {X 0,Y 270.166,Z 753.632,A -85,B 0,C 180,E1 -17686.751,E2 -17686.751} C_VEL
LIN {X 0,Y 270.222,Z 753.638,A -85,B 0,C 180,E1 -17691.283,E2 -17691.283} C_VEL
LIN {X 0,Y 270.215,Z 753.628,A -85,B 0,C 180,E1 -17695.096,E2 -17695.096} C_VEL
LIN {X 0,Y 270.267,Z 753.687,A -85,B 0,C 180,E1 -17698.809,E2 -17698.809} C_VEL
LIN {X 0,Y 272.079,Z 762.711,A -85,B 0,C 180,E1 -17702.71,E2 -17702.71} C_VEL
LIN {X 0,Y 273.305,Z 770.173,A -85,B 0,C 180,E1 -17705.705,E2 -17705.705} C_VEL
LIN {X 0,Y 273.025,Z 772.733,A -85,B 0,C 180,E1 -17706.585,E2 -17706.585} C_VEL
LIN {X 0,Y 273.748,Z 777.212,A -85,B 0,C 180,E1 -17706.855,E2 -17706.855} C_VEL
LIN {X 0,Y 277.434,Z 799.243,A -85,B 0,C 180,E1 -17707.781,E2 -17707.781} C_VEL
LIN {X 0,Y 279.095,Z 813.22,A -85,B 0,C 180,E1 -17708.298,E2 -17708.298} C_VEL
LIN {X 0,Y 278.148,Z 850.496,A -85,B 0,C 180,E1 -17709.284,E2 -17709.284} C_VEL
LIN {X 0,Y 277.429,Z 861.942,A -85,B 0,C 180,E1 -17709.825,E2 -17709.825} C_VEL
LIN {X 0,Y 276.364,Z 873.358,A -85,B 0,C 180,E1 -17710.695,E2 -17710.695} C_VEL
LIN {X 0,Y 275.389,Z 882.052,A -85,B 0,C 180,E1 -17711.59,E2 -17711.59} C_VEL
LIN {X 0,Y 274.271,Z 890.358,A -85,B 0,C 180,E1 -17712.67,E2 -17712.67} C_VEL
LIN {X 0,Y 273.08,Z 898.221,A -85,B 0,C 180,E1 -17713.939,E2 -17713.939} C_VEL
LIN {X 0,Y 271.825,Z 905.575,A -85,B 0,C 180,E1 -17715.399,E2 -17715.399} C_VEL
LIN {X 0,Y 270.66,Z 913.043,A -85,B 0,C 180,E1 -17717.249,E2 -17717.249} C_VEL
LIN {X 0,Y 269.677,Z 918.898,A -85,B 0,C 180,E1 -17719.109,E2 -17719.109} C_VEL
LIN {X 0,Y 269.006,Z 923.517,A -85,B 0,C 180,E1 -17720.981,E2 -17720.981} C_VEL
LIN {X 0,Y 268.636,Z 926.521,A -85,B 0,C 180,E1 -17722.484,E2 -17722.484} C_VEL
LIN {X 0,Y 268.318,Z 929.481,A -85,B 0,C 180,E1 -17724.457,E2 -17724.457} C_VEL
LIN {X 0,Y 268.186,Z 931.859,A -85,B 0,C 180,E1 -17726.996,E2 -17726.996} C_VEL
LIN {X 0,Y 268.19,Z 932.639,A -85,B 0,C 180,E1 -17728.498,E2 -17728.498} C_VEL
LIN {X 0,Y 268.201,Z 932.934,A -85,B 0,C 180,E1 -17730,E2 -17730} C_VEL
LIN {X 0,Y 268.19,Z 932.633,A -85,B 0,C 180,E1 -17731.502,E2 -17731.502} C_VEL
LIN {X 0,Y 268.186,Z 931.841,A -85,B 0,C 180,E1 -17733.004,E2 -17733.004} C_VEL
LIN {X 0,Y 268.316,Z 929.456,A -85,B 0,C 180,E1 -17735.539,E2 -17735.539} C_VEL
LIN {X 0,Y 268.636,Z 926.476,A -85,B 0,C 180,E1 -17737.516,E2 -17737.516} C_VEL
LIN {X 0,Y 269.248,Z 921.713,A -85,B 0,C 180,E1 -17739.768,E2 -17739.768} C_VEL
LIN {X 0,Y 270.034,Z 916.558,A -85,B 0,C 180,E1 -17741.637,E2 -17741.637} C_VEL
LIN {X 0,Y 270.863,Z 911.522,A -85,B 0,C 180,E1 -17743.122,E2 -17743.122} C_VEL
LIN {X 0,Y 271.823,Z 905.458,A -85,B 0,C 180,E1 -17744.601,E2 -17744.601} C_VEL
LIN {X 0,Y 273.053,Z 898.083,A -85,B 0,C 180,E1 -17746.063,E2 -17746.063} C_VEL
LIN {X 0,Y 274.276,Z 890.186,A -85,B 0,C 180,E1 -17747.33,E2 -17747.33} C_VEL
LIN {X 0,Y 275.415,Z 881.84,A -85,B 0,C 180,E1 -17748.408,E2 -17748.408} C_VEL
LIN {X 0,Y 276.527,Z 871.393,A -85,B 0,C 180,E1 -17749.465,E2 -17749.465} C_VEL
LIN {X 0,Y 277.541,Z 860.051,A -85,B 0,C 180,E1 -17750.249,E2 -17750.249} C_VEL
LIN {X 0,Y 278.111,Z 850.827,A -85,B 0,C 180,E1 -17750.679,E2 -17750.679} C_VEL
LIN {X 0,Y 278.858,Z 819.214,A -85,B 0,C 180,E1 -17751.53,E2 -17751.53} C_VEL
LIN {X 0,Y 278.912,Z 810.805,A -85,B 0,C 180,E1 -17751.754,E2 -17751.754} C_VEL
LIN {X 0,Y 275.13,Z 784.834,A -85,B 0,C 180,E1 -17752.782,E2 -17752.782} C_VEL
LIN {X 0,Y 273.037,Z 772.957,A -85,B 0,C 180,E1 -17753.348,E2 -17753.348} C_VEL
LIN {X 0,Y 273.303,Z 770.097,A -85,B 0,C 180,E1 -17754.295,E2 -17754.295} C_VEL
LIN {X 0,Y 272.096,Z 762.66,A -85,B 0,C 180,E1 -17757.288,E2 -17757.288} C_VEL
LIN {X 0,Y 270.29,Z 753.829,A -85,B 0,C 180,E1 -17761.042,E2 -17761.042} C_VEL
LIN {X 0,Y 270.205,Z 753.636,A -85,B 0,C 180,E1 -17763.107,E2 -17763.107} C_VEL
LIN {X 0,Y 270.238,Z 753.625,A -85,B 0,C 180,E1 -17766.738,E2 -17766.738} C_VEL
LIN {X 0,Y 270.174,Z 753.619,A -85,B 0,C 180,E1 -17770.566,E2 -17770.566} C_VEL
LIN {X 0,Y 270.157,Z 753.644,A -85,B 0,C 180,E1 -17774.619,E2 -17774.619} C_VEL
LIN {X 0,Y 270.2,Z 753.586,A -85,B 0,C 180,E1 -17778.964,E2 -17778.964} C_VEL
LIN {X 0,Y 270.245,Z 753.57,A -85,B 0,C 180,E1 -17781.381,E2 -17781.381} C_VEL
LIN {X 0,Y 270.216,Z 753.631,A -85,B 0,C 180,E1 -17785.097,E2 -17785.097} C_VEL
LIN {X 0,Y 270.201,Z 753.628,A -85,B 0,C 180,E1 -17789.131,E2 -17789.131} C_VEL
LIN {X 0,Y 270.264,Z 753.62,A -85,B 0,C 180,E1 -17792.146,E2 -17792.146} C_VEL
LIN {X 0,Y 270.278,Z 753.63,A -85,B 0,C 180,E1 -17795.519,E2 -17795.519} C_VEL
LIN {X 0,Y 270.303,Z 753.61,A -85,B 0,C 180,E1 -17800.245,E2 -17800.245} C_VEL
LIN {X 0,Y 270.404,Z 753.606,A -85,B 0,C 180,E1 -17804.936,E2 -17804.936} C_VEL
LIN {X 0,Y 270.443,Z 753.594,A -85,B 0,C 180,E1 -17809.519,E2 -17809.519} C_VEL
LIN {X 0,Y 270.604,Z 753.591,A -85,B 0,C 180,E1 -17812.539,E2 -17812.539} C_VEL
LIN {X 0,Y 270.789,Z 753.536,A -85,B 0,C 180,E1 -17818.513,E2 -17818.513} C_VEL
LIN {X 0,Y 270.792,Z 753.562,A -85,B 0,C 180,E1 -17821.487,E2 -17821.487} C_VEL
LIN {X 0,Y 270.613,Z 753.554,A -85,B 0,C 180,E1 -17827.461,E2 -17827.461} C_VEL
LIN {X 0,Y 270.443,Z 753.6,A -85,B 0,C 180,E1 -17830.481,E2 -17830.481} C_VEL
LIN {X 0,Y 270.375,Z 753.605,A -85,B 0,C 180,E1 -17835.066,E2 -17835.066} C_VEL
LIN {X 0,Y 270.281,Z 753.624,A -85,B 0,C 180,E1 -17839.757,E2 -17839.757} C_VEL
LIN {X 0,Y 270.239,Z 753.618,A -85,B 0,C 180,E1 -17844.589,E2 -17844.589} C_VEL
LIN {X 0,Y 270.271,Z 753.624,A -85,B 0,C 180,E1 -17847.909,E2 -17847.909} C_VEL
LIN {X 0,Y 270.185,Z 753.635,A -85,B 0,C 180,E1 -17851.348,E2 -17851.348} C_VEL
LIN {X 0,Y 270.203,Z 753.629,A -85,B 0,C 180,E1 -17854.905,E2 -17854.905} C_VEL
LIN {X 0,Y 270.199,Z 753.631,A -85,B 0,C 180,E1 -17858.71,E2 -17858.71} C_VEL
LIN {X 0,Y 270.172,Z 753.583,A -85,B 0,C 180,E1 -17862.558,E2 -17862.558} C_VEL
LIN {X 0,Y 270.166,Z 753.642,A -85,B 0,C 180,E1 -17866.751,E2 -17866.751} C_VEL
LIN {X 0,Y 270.175,Z 753.631,A -85,B 0,C 180,E1 -17869.434,E2 -17869.434} C_VEL
LIN {X 0,Y 270.226,Z 753.627,A -85,B 0,C 180,E1 -17873.731,E2 -17873.731} C_VEL
LIN {X 0,Y 270.203,Z 753.629,A -85,B 0,C 180,E1 -17876.892,E2 -17876.892} C_VEL
LIN {X 0,Y 270.184,Z 753.642,A -85,B 0,C 180,E1 -17880.381,E2 -17880.381} C_VEL
LIN {X 0,Y 270.299,Z 753.736,A -85,B 0,C 180,E1 -17884.286,E2 -17884.286} C_VEL
LIN {X 0,Y 271.245,Z 758.698,A -85,B 0,C 180,E1 -17886.523,E2 -17886.523} C_VEL
LIN {X 0,Y 272.66,Z 762.652,A -85,B 0,C 180,E1 -17886.839,E2 -17886.839} C_VEL
LIN {X 0,Y 276.661,Z 773.548,A -85,B 0,C 180,E1 -17887.498,E2 -17887.498} C_VEL
LIN {X 0,Y 279.537,Z 789.13,A -85,B 0,C 180,E1 -17888.168,E2 -17888.168} C_VEL
LIN {X 0,Y 278.441,Z 834.517,A -85,B 0,C 180,E1 -17889.355,E2 -17889.355} C_VEL
LIN {X 0,Y 278.054,Z 844.247,A -85,B 0,C 180,E1 -17889.808,E2 -17889.808} C_VEL
LIN {X 0,Y 277.126,Z 855.303,A -85,B 0,C 180,E1 -17890.558,E2 -17890.558} C_VEL
LIN {X 0,Y 276.106,Z 866.089,A -85,B 0,C 180,E1 -17891.64,E2 -17891.64} C_VEL
LIN {X 0,Y 274.911,Z 874.471,A -85,B 0,C 180,E1 -17892.711,E2 -17892.711} C_VEL
LIN {X 0,Y 273.85,Z 882.378,A -85,B 0,C 180,E1 -17893.985,E2 -17893.985} C_VEL
LIN {X 0,Y 272.997,Z 888.055,A -85,B 0,C 180,E1 -17895.082,E2 -17895.082} C_VEL
LIN {X 0,Y 271.916,Z 894.396,A -85,B 0,C 180,E1 -17896.549,E2 -17896.549} C_VEL
LIN {X 0,Y 270.974,Z 899.665,A -85,B 0,C 180,E1 -17898.025,E2 -17898.025} C_VEL
LIN {X 0,Y 270.208,Z 904.062,A -85,B 0,C 180,E1 -17899.51,E2 -17899.51} C_VEL
LIN {X 0,Y 269.418,Z 909.229,A -85,B 0,C 180,E1 -17901.751,E2 -17901.751} C_VEL
LIN {X 0,Y 268.994,Z 911.708,A -85,B 0,C 180,E1 -17903.135,E2 -17903.135} C_VEL
LIN {X 0,Y 268.563,Z 914.781,A -85,B 0,C 180,E1 -17905.497,E2 -17905.497} C_VEL
LIN {X 0,Y 268.387,Z 916.047,A -85,B 0,C 180,E1 -17906.998,E2 -17906.998} C_VEL
LIN {X 0,Y 268.24,Z 916.845,A -85,B 0,C 180,E1 -17908.499,E2 -17908.499} C_VEL
LIN {X 0,Y 268.209,Z 917.149,A -85,B 0,C 180,E1 -17910,E2 -17910} C_VEL
LIN {X 0,Y 268.238,Z 916.87,A -85,B 0,C 180,E1 -17911.501,E2 -17911.501} C_VEL
LIN {X 0,Y 268.382,Z 916.121,A -85,B 0,C 180,E1 -17913.002,E2 -17913.002} C_VEL
LIN {X 0,Y 268.558,Z 914.906,A -85,B 0,C 180,E1 -17914.503,E2 -17914.503} C_VEL
LIN {X 0,Y 268.808,Z 913.202,A -85,B 0,C 180,E1 -17916.003,E2 -17916.003} C_VEL
LIN {X 0,Y 269.367,Z 909.464,A -85,B 0,C 180,E1 -17918.25,E2 -17918.25} C_VEL
LIN {X 0,Y 270.152,Z 904.36,A -85,B 0,C 180,E1 -17920.492,E2 -17920.492} C_VEL
LIN {X 0,Y 271.177,Z 898.862,A -85,B 0,C 180,E1 -17922.346,E2 -17922.346} C_VEL
LIN {X 0,Y 272.426,Z 891.95,A -85,B 0,C 180,E1 -17924.187,E2 -17924.187} C_VEL
LIN {X 0,Y 273.627,Z 884.015,A -85,B 0,C 180,E1 -17925.837,E2 -17925.837} C_VEL
LIN {X 0,Y 274.708,Z 876.446,A -85,B 0,C 180,E1 -17927.11,E2 -17927.11} C_VEL
LIN {X 0,Y 275.815,Z 868.505,A -85,B 0,C 180,E1 -17928.188,E2 -17928.188} C_VEL
LIN {X 0,Y 276.77,Z 860.298,A -85,B 0,C 180,E1 -17929.083,E2 -17929.083} C_VEL
LIN {X 0,Y 277.592,Z 851.97,A -85,B 0,C 180,E1 -17929.793,E2 -17929.793} C_VEL
LIN {X 0,Y 278.131,Z 842.955,A -85,B 0,C 180,E1 -17930.379,E2 -17930.379} C_VEL
LIN {X 0,Y 278.526,Z 833.599,A -85,B 0,C 180,E1 -17930.791,E2 -17930.791} C_VEL
LIN {X 0,Y 279.514,Z 787.997,A -85,B 0,C 180,E1 -17931.983,E2 -17931.983} C_VEL
LIN {X 0,Y 276.507,Z 773.046,A -85,B 0,C 180,E1 -17932.649,E2 -17932.649} C_VEL
LIN {X 0,Y 271.36,Z 759.001,A -85,B 0,C 180,E1 -17933.542,E2 -17933.542} C_VEL
LIN {X 0,Y 271.053,Z 757.595,A -85,B 0,C 180,E1 -17933.992,E2 -17933.992} C_VEL
LIN {X 0,Y 270.278,Z 753.709,A -85,B 0,C 180,E1 -17935.923,E2 -17935.923} C_VEL
LIN {X 0,Y 270.184,Z 753.643,A -85,B 0,C 180,E1 -17939.619,E2 -17939.619} C_VEL
LIN {X 0,Y 270.216,Z 753.634,A -85,B 0,C 180,E1 -17943.666,E2 -17943.666} C_VEL
LIN {X 0,Y 270.217,Z 753.622,A -85,B 0,C 180,E1 -17946.741,E2 -17946.741} C_VEL
LIN {X 0,Y 270.17,Z 753.636,A -85,B 0,C 180,E1 -17951.028,E2 -17951.028} C_VEL
LIN {X 0,Y 270.153,Z 753.629,A -85,B 0,C 180,E1 -17954.62,E2 -17954.62} C_VEL
LIN {X 0,Y 270.172,Z 753.584,A -85,B 0,C 180,E1 -17957.442,E2 -17957.442} C_VEL
LIN {X 0,Y 270.208,Z 753.629,A -85,B 0,C 180,E1 -17961.374,E2 -17961.374} C_VEL
LIN {X 0,Y 270.203,Z 753.63,A -85,B 0,C 180,E1 -17965.095,E2 -17965.095} C_VEL
LIN {X 0,Y 270.202,Z 753.637,A -85,B 0,C 180,E1 -17969.131,E2 -17969.131} C_VEL
LIN {X 0,Y 270.264,Z 753.626,A -85,B 0,C 180,E1 -17972.146,E2 -17972.146} C_VEL
LIN {X 0,Y 270.238,Z 753.618,A -85,B 0,C 180,E1 -17975.538,E2 -17975.538} C_VEL
LIN {X 0,Y 270.298,Z 753.622,A -85,B 0,C 180,E1 -17980.244,E2 -17980.244} C_VEL
LIN {X 0,Y 270.375,Z 753.604,A -85,B 0,C 180,E1 -17984.934,E2 -17984.934} C_VEL
LIN {X 0,Y 270.464,Z 753.595,A -85,B 0,C 180,E1 -17989.759,E2 -17989.759} C_VEL
LIN {X 0,Y 270.613,Z 753.554,A -85,B 0,C 180,E1 -17992.539,E2 -17992.539} C_VEL
LIN {X 0,Y 270.497,Z 753.595,A -85,B 0,C 180,E1 -17996.19,E2 -17996.19} C_VEL
LIN {X 0,Y 269.973,Z 753.67,A -85,B 0,C 180,E1 -17997.435,E2 -17997.435} C_VEL
LIN {X 0,Y 268.482,Z 753.85,A -85,B 0,C 180,E1 -17998.659,E2 -17998.659} C_VEL
LIN {X 0,Y 264.793,Z 754.286,A -85,B 0,C 180,E1 -18001.118,E2 -18001.118} C_VEL
LIN {X 0,Y 263.694,Z 754.415,A -85,B 0,C 180,E1 -18002.397,E2 -18002.397} C_VEL
LIN {X 0,Y 263.58,Z 754.43,A -85,B 0,C 180,E1 -18002.831,E2 -18002.831} C_VEL
LIN {X 0,Y 263.566,Z 754.468,A -85,B 0,C 180,E1 -18007.662,E2 -18007.662} C_VEL
LIN {X 0,Y 263.375,Z 754.469,A -85,B 0,C 180,E1 -18010.765,E2 -18010.765} C_VEL
LIN {X 0,Y 263.352,Z 754.487,A -85,B 0,C 180,E1 -18015.478,E2 -18015.478} C_VEL
LIN {X 0,Y 263.265,Z 754.481,A -85,B 0,C 180,E1 -18020.306,E2 -18020.306} C_VEL
LIN {X 0,Y 263.209,Z 754.51,A -85,B 0,C 180,E1 -18025.291,E2 -18025.291} C_VEL
LIN {X 0,Y 263.166,Z 754.496,A -85,B 0,C 180,E1 -18028.731,E2 -18028.731} C_VEL
LIN {X 0,Y 263.134,Z 754.52,A -85,B 0,C 180,E1 -18032.288,E2 -18032.288} C_VEL
LIN {X 0,Y 263.189,Z 754.491,A -85,B 0,C 180,E1 -18035.978,E2 -18035.978} C_VEL
LIN {X 0,Y 263.139,Z 754.453,A -85,B 0,C 180,E1 -18039.866,E2 -18039.866} C_VEL
LIN {X 0,Y 263.129,Z 754.518,A -85,B 0,C 180,E1 -18043.983,E2 -18043.983} C_VEL
LIN {X 0,Y 263.124,Z 754.494,A -85,B 0,C 180,E1 -18048.406,E2 -18048.406} C_VEL
LIN {X 0,Y 263.166,Z 754.518,A -85,B 0,C 180,E1 -18052.104,E2 -18052.104} C_VEL
LIN {X 0,Y 263.184,Z 754.515,A -85,B 0,C 180,E1 -18055.89,E2 -18055.89} C_VEL
LIN {X 0,Y 263.191,Z 754.647,A -85,B 0,C 180,E1 -18058.416,E2 -18058.416} C_VEL
LIN {X 0,Y 265.062,Z 763.551,A -85,B 0,C 180,E1 -18062.354,E2 -18062.354} C_VEL
LIN {X 0,Y 266.319,Z 771.017,A -85,B 0,C 180,E1 -18065.441,E2 -18065.441} C_VEL
LIN {X 0,Y 266.273,Z 772.87,A -85,B 0,C 180,E1 -18066.002,E2 -18066.002} C_VEL
LIN {X 0,Y 270.073,Z 794.872,A -85,B 0,C 180,E1 -18067.024,E2 -18067.024} C_VEL
LIN {X 0,Y 272.503,Z 813.913,A -85,B 0,C 180,E1 -18067.77,E2 -18067.77} C_VEL
LIN {X 0,Y 271.53,Z 850.303,A -85,B 0,C 180,E1 -18068.755,E2 -18068.755} C_VEL
LIN {X 0,Y 270.796,Z 861.734,A -85,B 0,C 180,E1 -18069.308,E2 -18069.308} C_VEL
LIN {X 0,Y 269.688,Z 873.155,A -85,B 0,C 180,E1 -18070.198,E2 -18070.198} C_VEL
LIN {X 0,Y 268.649,Z 881.847,A -85,B 0,C 180,E1 -18071.111,E2 -18071.111} C_VEL
LIN {X 0,Y 267.502,Z 890.152,A -85,B 0,C 180,E1 -18072.217,E2 -18072.217} C_VEL
LIN {X 0,Y 266.258,Z 898.015,A -85,B 0,C 180,E1 -18073.516,E2 -18073.516} C_VEL
LIN {X 0,Y 264.944,Z 905.369,A -85,B 0,C 180,E1 -18075.011,E2 -18075.011} C_VEL
LIN {X 0,Y 263.731,Z 912.835,A -85,B 0,C 180,E1 -18076.908,E2 -18076.908} C_VEL
LIN {X 0,Y 262.53,Z 919.652,A -85,B 0,C 180,E1 -18079.199,E2 -18079.199} C_VEL
LIN {X 0,Y 261.751,Z 924.835,A -85,B 0,C 180,E1 -18081.508,E2 -18081.508} C_VEL
LIN {X 0,Y 261.296,Z 928.644,A -85,B 0,C 180,E1 -18083.824,E2 -18083.824} C_VEL
LIN {X 0,Y 261.145,Z 930.395,A -85,B 0,C 180,E1 -18085.369,E2 -18085.369} C_VEL
LIN {X 0,Y 261.103,Z 931.65,A -85,B 0,C 180,E1 -18086.914,E2 -18086.914} C_VEL
LIN {X 0,Y 261.117,Z 932.431,A -85,B 0,C 180,E1 -18088.458,E2 -18088.458} C_VEL
LIN {X 0,Y 261.126,Z 932.725,A -85,B 0,C 180,E1 -18090,E2 -18090} C_VEL
